C03639=1038.080,62.788,410.793,169.407,39.489,157.422
C03640=1038.074,62.538,410.811,169.405,39.489,157.422
C03641=1038.068,62.289,410.828,169.403,39.488,157.421
C03642=1038.061,62.040,410.846,169.401,39.489,157.421
C03643=1038.055,61.791,410.864,169.399,39.488,157.421
C03644=1038.048,61.541,410.881,169.397,39.488,157.421
C03645=1038.042,61.292,410.899,169.394,39.488,157.421
C03646=1038.035,61.005,410.919,169.392,39.488,157.421
C03647=1038.028,60.719,410.939,169.390,39.487,157.421
C03648=1038.019,60.433,410.959,169.387,39.488,157.421
C03649=1038.012,60.147,410.979,169.385,39.487,157.421
C03650=1038.006,59.897,410.997,169.383,39.487,157.421
C03651=1037.999,59.648,411.014,169.381,39.487,157.420
C03652=1037.994,59.399,411.031,169.379,39.487,157.420
C03653=1037.987,59.150,411.049,169.377,39.487,157.420
C03654=1037.980,58.900,411.066,169.375,39.487,157.420
C03655=1037.974,58.650,411.084,169.373,39.486,157.420
C03656=1037.968,58.402,411.101,169.370,39.486,157.420
C03657=1037.961,58.152,411.118,169.368,39.486,157.420
C03658=1037.955,57.902,411.136,169.366,39.486,157.420
C03659=1037.949,57.654,411.153,169.364,39.486,157.420
C03660=1037.942,57.404,411.171,169.362,39.486,157.419
C03661=1037.936,57.155,411.188,169.360,39.485,157.419
C03662=1037.929,56.906,411.206,169.358,39.485,157.419
C03663=1037.923,56.656,411.223,169.357,39.485,157.419
C03664=1037.917,56.407,411.240,169.355,39.485,157.419
C03665=1037.910,56.158,411.258,169.353,39.485,157.419
C03666=1037.904,55.908,411.276,169.351,39.485,157.419
C03667=1037.898,55.660,411.293,169.349,39.484,157.419
C03668=1037.891,55.410,411.310,169.347,39.484,157.419
C03669=1037.885,55.161,411.328,169.344,39.484,157.419
C03670=1037.878,54.912,411.345,169.342,39.483,157.418
C03671=1037.872,54.662,411.362,169.340,39.484,157.418
C03672=1037.866,54.413,411.380,169.338,39.483,157.418
C03673=1037.860,54.163,411.396,169.336,39.483,157.418
C03674=1037.853,53.914,411.413,169.334,39.483,157.418
C03675=1037.847,53.665,411.431,169.332,39.483,157.418
C03676=1037.840,53.415,411.449,169.330,39.482,157.418
C03677=1037.834,53.166,411.466,169.328,39.483,157.418
C03678=1037.828,52.917,411.484,169.326,39.482,157.418
C03679=1037.822,52.668,411.501,169.324,39.482,157.418
C03680=1037.815,52.418,411.517,169.321,39.482,157.417
C03681=1037.810,52.169,411.535,169.319,39.481,157.417
C03682=1037.803,51.919,411.552,169.317,39.481,157.417
C03683=1037.796,51.671,411.569,169.315,39.481,157.417
C03684=1037.790,51.421,411.587,169.313,39.481,157.417
C03685=1037.784,51.172,411.604,169.311,39.481,157.417
C03686=1037.778,50.922,411.621,169.309,39.481,157.417
C03687=1037.771,50.672,411.639,169.307,39.480,157.417
C03688=1037.765,50.424,411.655,169.305,39.480,157.417
C03689=1037.758,50.174,411.673,169.303,39.480,157.416
C03690=1037.753,49.925,411.690,169.300,39.479,157.416
C03691=1037.746,49.675,411.707,169.298,39.480,157.416
C03692=1037.740,49.427,411.724,169.296,39.479,157.416
C03693=1037.734,49.177,411.742,169.294,39.479,157.416
C03694=1037.728,48.927,411.758,169.293,39.479,157.416
C03695=1037.721,48.678,411.776,169.291,39.478,157.416
C03696=1037.716,48.429,411.793,169.289,39.478,157.416
C03697=1037.709,48.180,411.810,169.287,39.478,157.415
C03698=1037.703,47.930,411.827,169.285,39.478,157.415
C03699=1037.697,47.681,411.844,169.283,39.478,157.415
C03700=1037.690,47.432,411.862,169.280,39.477,157.415
C03701=1037.684,47.182,411.878,169.278,39.477,157.415
C03702=1037.678,46.933,411.896,169.276,39.477,157.415
C03703=1037.672,46.684,411.913,169.274,39.477,157.415
C03704=1037.665,46.434,411.929,169.272,39.476,157.415
C03705=1037.659,46.185,411.946,169.270,39.476,157.415
C03706=1037.653,45.935,411.964,169.268,39.476,157.415
C03707=1037.647,45.686,411.981,169.266,39.476,157.414
C03708=1037.641,45.437,411.998,169.264,39.476,157.414
C03709=1037.635,45.188,412.015,169.262,39.475,157.414
C03710=1037.627,44.901,412.034,169.260,39.475,157.414
C03711=1037.620,44.614,412.054,169.258,39.475,157.414
C03712=1037.613,44.328,412.074,169.254,39.474,157.414
C03713=1037.606,44.042,412.093,169.252,39.474,157.414
C03714=1037.600,43.792,412.110,169.250,39.474,157.414
C03715=1037.594,43.542,412.127,169.248,39.474,157.413
C03716=1037.588,43.293,412.144,169.246,39.473,157.413
C03717=1037.582,43.044,412.161,169.244,39.473,157.413
C03718=1037.575,42.795,412.178,169.242,39.473,157.413
C03719=1037.569,42.545,412.194,169.240,39.473,157.413
C03720=1037.563,42.296,412.211,169.238,39.472,157.413
C03721=1037.556,42.046,412.228,169.236,39.473,157.413
C03722=1037.550,41.797,412.245,169.233,39.472,157.413
C03723=1037.544,41.548,412.261,169.231,39.472,157.413
C03724=1037.537,41.299,412.278,169.229,39.472,157.412
C03725=1037.531,41.049,412.295,169.227,39.472,157.412
C03726=1037.524,40.800,412.312,169.225,39.471,157.412
C03727=1037.518,40.550,412.328,169.223,39.472,157.412
C03728=1037.512,40.302,412.345,169.221,39.471,157.412
C03729=1037.505,40.052,412.362,169.219,39.471,157.412
C03730=1037.499,39.802,412.378,169.217,39.471,157.412
C03731=1037.493,39.553,412.395,169.215,39.471,157.412
C03732=1037.487,39.303,412.412,169.213,39.470,157.412
C03733=1037.481,39.055,412.429,169.211,39.471,157.412
C03734=1037.475,38.804,412.446,169.208,39.470,157.411
C03735=1037.469,38.555,412.462,169.206,39.470,157.411
C03736=1037.462,38.306,412.479,169.204,39.470,157.411
C03737=1037.456,38.056,412.496,169.202,39.470,157.411
C03738=1037.450,37.807,412.512,169.200,39.469,157.411
C03739=1037.444,37.558,412.529,169.198,39.470,157.411
C03740=1037.437,37.308,412.546,169.196,39.469,157.411
C03741=1037.430,37.059,412.561,169.194,39.469,157.411
C03742=1037.424,36.810,412.578,169.192,39.469,157.411
C03743=1037.418,36.560,412.595,169.190,39.469,157.411
C03744=1037.412,36.311,412.611,169.188,39.469,157.411
C03745=1037.405,36.061,412.628,169.186,39.469,157.410
C03746=1037.398,35.813,412.644,169.184,39.469,157.410
C03747=1037.392,35.563,412.660,169.182,39.469,157.410
C03748=1037.386,35.313,412.677,169.179,39.468,157.410
C03749=1037.380,35.064,412.693,169.177,39.469,157.410
C03750=1037.373,34.815,412.710,169.175,39.468,157.410
C03751=1037.366,34.565,412.726,169.173,39.468,157.410
C03752=1037.360,34.316,412.743,169.171,39.468,157.410
C03753=1037.354,34.067,412.759,169.169,39.468,157.410
C03754=1037.348,33.817,412.775,169.167,39.468,157.410
C03755=1037.341,33.568,412.792,169.165,39.468,157.409
C03756=1037.335,33.319,412.808,169.163,39.468,157.409
C03757=1037.329,33.070,412.824,169.161,39.467,157.409
C03758=1037.322,32.819,412.841,169.159,39.467,157.409
C03759=1037.316,32.570,412.857,169.157,39.468,157.409
C03760=1037.309,32.321,412.873,169.155,39.467,157.409
C03761=1037.304,32.072,412.889,169.153,39.467,157.409
C03762=1037.297,31.822,412.906,169.150,39.467,157.409
C03763=1037.291,31.573,412.923,169.147,39.467,157.409
C03764=1037.285,31.324,412.939,169.145,39.466,157.409
C03765=1037.278,31.075,412.955,169.143,39.467,157.409
C03766=1037.272,30.825,412.971,169.141,39.467,157.409
C03767=1037.266,30.575,412.987,169.139,39.466,157.408
C03768=1037.260,30.326,413.004,169.137,39.466,157.408
C03769=1037.253,30.077,413.019,169.135,39.466,157.408
C03770=1037.246,29.827,413.036,169.133,39.466,157.408
C03771=1037.240,29.577,413.052,169.131,39.466,157.408
C03772=1037.234,29.328,413.069,169.129,39.466,157.408
C03773=1037.227,29.080,413.085,169.127,39.466,157.408
C03774=1037.221,28.792,413.104,169.124,39.465,157.408
C03775=1037.213,28.505,413.122,169.121,39.465,157.408
C03776=1037.206,28.219,413.141,169.119,39.465,157.407
C03777=1037.199,27.932,413.159,169.117,39.465,157.407
C03778=1037.193,27.683,413.175,169.115,39.465,157.407
C03779=1037.185,27.433,413.191,169.113,39.465,157.407
C03780=1037.179,27.184,413.208,169.111,39.464,157.407
C03781=1037.174,26.935,413.224,169.109,39.465,157.407
C03782=1037.167,26.686,413.239,169.106,39.465,157.407
C03783=1037.161,26.436,413.256,169.104,39.464,157.407
C03784=1037.154,26.186,413.272,169.102,39.464,157.407
C03785=1037.148,25.937,413.288,169.100,39.465,157.407
C03786=1037.142,25.688,413.304,169.098,39.464,157.407
C03787=1037.135,25.439,413.320,169.096,39.464,157.407
C03788=1037.129,25.189,413.335,169.094,39.464,157.407
C03789=1037.122,24.939,413.351,169.091,39.464,157.406
C03790=1037.116,24.690,413.368,169.089,39.464,157.406
C03791=1037.109,24.441,413.383,169.087,39.464,157.406
C03792=1037.103,24.191,413.400,169.085,39.464,157.406
C03793=1037.097,23.942,413.415,169.083,39.464,157.406
C03794=1037.091,23.693,413.432,169.081,39.464,157.406
C03795=1037.084,23.443,413.447,169.079,39.464,157.406
C03796=1037.078,23.193,413.463,169.076,39.464,157.406
C03797=1037.071,22.944,413.479,169.074,39.464,157.406
C03798=1037.065,22.695,413.495,169.072,39.463,157.406
C03799=1037.059,22.446,413.511,169.070,39.464,157.406
C03800=1037.053,22.196,413.526,169.068,39.463,157.405
C03801=1037.046,21.947,413.542,169.066,39.463,157.405
C03802=1037.040,21.697,413.558,169.064,39.463,157.405
C03803=1037.033,21.448,413.574,169.062,39.463,157.405
C03804=1037.027,21.198,413.590,169.060,39.463,157.405
C03805=1037.021,20.949,413.605,169.057,39.463,157.405
C03806=1037.015,20.699,413.622,169.055,39.463,157.405
C03807=1037.008,20.450,413.637,169.053,39.463,157.405
C03808=1037.002,20.201,413.654,169.051,39.462,157.405
C03809=1036.996,19.951,413.669,169.048,39.463,157.405
C03810=1036.990,19.702,413.685,169.046,39.463,157.405
C03811=1036.983,19.453,413.700,169.044,39.462,157.404
C03812=1036.977,19.202,413.716,169.042,39.462,157.404
C03813=1036.970,18.953,413.732,169.040,39.463,157.404
C03814=1036.963,18.704,413.748,169.038,39.463,157.404
C03815=1036.958,18.454,413.763,169.036,39.462,157.404
C03816=1036.951,18.205,413.779,169.034,39.462,157.404
C03817=1036.945,17.956,413.795,169.032,39.463,157.404
C03818=1036.939,17.706,413.810,169.030,39.462,157.404
C03819=1036.932,17.457,413.826,169.027,39.462,157.404
C03820=1036.926,17.207,413.841,169.025,39.463,157.404
C03821=1036.920,16.958,413.857,169.022,39.462,157.404
C03822=1036.913,16.709,413.873,169.020,39.462,157.404
C03823=1036.907,16.459,413.888,169.018,39.462,157.404
C03824=1036.901,16.210,413.904,169.016,39.462,157.403
C03825=1036.894,15.960,413.919,169.014,39.462,157.403
C03826=1036.888,15.711,413.935,169.012,39.462,157.403
C03827=1036.882,15.462,413.951,169.010,39.462,157.403
C03828=1036.875,15.212,413.966,169.007,39.462,157.403
C03829=1036.869,14.963,413.982,169.005,39.462,157.403
C03830=1036.862,14.713,413.997,169.003,39.462,157.403
C03831=1036.856,14.463,414.013,169.001,39.462,157.403
C03832=1036.850,14.214,414.028,168.999,39.462,157.403
C03833=1036.843,13.965,414.044,168.997,39.462,157.403
C03834=1036.837,13.715,414.059,168.995,39.461,157.403
C03835=1036.830,13.466,414.075,168.993,39.462,157.403
C03836=1036.825,13.216,414.090,168.990,39.462,157.403
C03837=1036.818,12.967,414.106,168.988,39.462,157.403
C03838=1036.811,12.681,414.123,168.986,39.462,157.402
C03839=1036.803,12.396,414.141,168.982,39.462,157.402
C03840=1036.796,12.111,414.158,168.980,39.462,157.402
C03841=1036.789,11.826,414.176,168.977,39.462,157.402
C03842=1036.782,11.576,414.190,168.975,39.462,157.402
C03843=1036.776,11.327,414.205,168.973,39.462,157.402
C03844=1036.769,11.078,414.221,168.971,39.462,157.402
C03845=1036.763,10.828,414.236,168.969,39.462,157.402
C03846=1036.756,10.579,414.252,168.967,39.462,157.402
C03847=1036.750,10.329,414.267,168.964,39.463,157.402
C03848=1036.743,10.080,414.282,168.962,39.463,157.402
C03849=1036.737,9.830,414.298,168.960,39.462,157.402
C03850=1036.731,9.581,414.313,168.958,39.462,157.402
C03851=1036.725,9.331,414.328,168.956,39.462,157.402
C03852=1036.718,9.082,414.343,168.954,39.463,157.402
C03853=1036.712,8.832,414.358,168.952,39.463,157.401
C03854=1036.705,8.583,414.373,168.949,39.462,157.401
C03855=1036.699,8.333,414.388,168.947,39.463,157.401
C03856=1036.692,8.084,414.404,168.945,39.463,157.401
C03857=1036.686,7.834,414.419,168.943,39.463,157.401
C03858=1036.679,7.585,414.434,168.941,39.463,157.401
C03859=1036.673,7.335,414.449,168.938,39.462,157.401
C03860=1036.666,7.086,414.464,168.935,39.463,157.401
C03861=1036.660,6.836,414.479,168.933,39.463,157.401
C03862=1036.655,6.587,414.494,168.931,39.463,157.401
C03863=1036.648,6.337,414.509,168.929,39.463,157.401
C03864=1036.642,6.088,414.525,168.927,39.463,157.401
C03865=1036.635,5.839,414.540,168.925,39.463,157.401
C03866=1036.629,5.589,414.555,168.922,39.463,157.401
C03867=1036.623,5.339,414.570,168.920,39.463,157.400
C03868=1036.616,5.090,414.586,168.918,39.463,157.400
C03869=1036.610,4.841,414.601,168.916,39.463,157.400
C03870=1036.603,4.591,414.615,168.914,39.463,157.400
C03871=1036.597,4.342,414.630,168.912,39.463,157.400
C03872=1036.591,4.092,414.645,168.909,39.463,157.400
C03873=1036.585,3.843,414.660,168.907,39.463,157.400
C03874=1036.578,3.594,414.676,168.905,39.463,157.400
C03875=1036.572,3.344,414.691,168.903,39.463,157.400
C03876=1036.565,3.094,414.706,168.901,39.463,157.400
C03877=1036.559,2.845,414.720,168.898,39.463,157.400
C03878=1036.553,2.596,414.735,168.896,39.463,157.400
C03879=1036.547,2.346,414.750,168.894,39.463,157.400
C03880=1036.540,2.097,414.765,168.892,39.463,157.400
C03881=1036.534,1.847,414.780,168.889,39.463,157.399
C03882=1036.527,1.597,414.795,168.887,39.463,157.399
C03883=1036.521,1.349,414.810,168.884,39.463,157.399
C03884=1036.515,1.099,414.825,168.882,39.463,157.399
C03885=1036.509,0.849,414.841,168.880,39.463,157.399
C03886=1036.503,0.600,414.856,168.878,39.463,157.399
C03887=1036.497,0.350,414.870,168.876,39.463,157.399
C03888=1036.491,0.101,414.885,168.874,39.463,157.399
C03889=1036.484,-0.149,414.900,168.871,39.464,157.399
C03890=1036.478,-0.398,414.915,168.869,39.463,157.399
C03891=1036.472,-0.648,414.930,168.867,39.463,157.399
C03892=1036.466,-0.897,414.944,168.865,39.463,157.399
C03893=1036.460,-1.147,414.959,168.863,39.463,157.399
C03894=1036.453,-1.396,414.974,168.860,39.463,157.398
C03895=1036.447,-1.646,414.989,168.858,39.463,157.398
C03896=1036.441,-1.895,415.004,168.856,39.464,157.398
C03897=1036.435,-2.145,415.019,168.854,39.463,157.398
C03898=1036.428,-2.394,415.034,168.852,39.463,157.398
C03899=1036.422,-2.644,415.049,168.849,39.463,157.398
C03900=1036.416,-2.893,415.063,168.846,39.464,157.398
C03901=1036.410,-3.142,415.078,168.844,39.463,157.398
C03902=1036.399,-3.564,415.103,168.840,39.463,157.398
C03903=1036.388,-3.986,415.128,168.837,39.464,157.398
C03904=1036.380,-4.308,415.147,168.834,39.464,157.398
C03905=1036.372,-4.630,415.165,168.831,39.464,157.398
C03906=1036.364,-4.952,415.184,168.828,39.464,157.398
C03907=1036.355,-5.275,415.203,168.825,39.464,157.397
C03908=1036.349,-5.524,415.217,168.823,39.464,157.397
C03909=1036.342,-5.773,415.232,168.820,39.464,157.397
C03910=1036.336,-6.023,415.246,168.818,39.464,157.397
C03911=1036.330,-6.272,415.261,168.816,39.465,157.397
C03912=1036.323,-6.522,415.275,168.814,39.465,157.397
C03913=1036.317,-6.771,415.290,168.811,39.465,157.397
C03914=1036.311,-7.021,415.304,168.809,39.465,157.397
C03915=1036.304,-7.270,415.318,168.807,39.465,157.397
C03916=1036.298,-7.520,415.333,168.805,39.465,157.397
C03917=1036.291,-7.769,415.348,168.802,39.466,157.397
C03918=1036.285,-8.019,415.361,168.800,39.466,157.397
C03919=1036.279,-8.268,415.376,168.798,39.466,157.397
C03920=1036.272,-8.518,415.391,168.796,39.466,157.397
C03921=1036.266,-8.767,415.404,168.793,39.466,157.397
C03922=1036.260,-9.017,415.419,168.791,39.466,157.397
C03923=1036.253,-9.267,415.434,168.789,39.466,157.397
C03924=1036.247,-9.516,415.448,168.787,39.466,157.397
C03925=1036.241,-9.766,415.463,168.784,39.466,157.397
C03926=1036.234,-10.015,415.478,168.782,39.467,157.396
C03927=1036.228,-10.264,415.491,168.779,39.467,157.396
C03928=1036.222,-10.514,415.506,168.777,39.467,157.396
C03929=1036.215,-10.763,415.520,168.774,39.467,157.396
C03930=1036.209,-11.013,415.534,168.772,39.467,157.396
C03931=1036.203,-11.263,415.549,168.770,39.467,157.396
C03932=1036.196,-11.511,415.563,168.767,39.468,157.396
C03933=1036.190,-11.762,415.577,168.765,39.467,157.396
C03934=1036.185,-12.011,415.592,168.763,39.467,157.396
C03935=1036.178,-12.260,415.605,168.761,39.467,157.396
C03936=1036.171,-12.510,415.620,168.758,39.468,157.396
C03937=1036.166,-12.760,415.634,168.756,39.468,157.396
C03938=1036.159,-13.009,415.648,168.754,39.468,157.396
C03939=1036.153,-13.258,415.663,168.752,39.468,157.396
C03940=1036.146,-13.508,415.677,168.749,39.468,157.396
C03941=1036.140,-13.758,415.692,168.747,39.468,157.396
C03942=1036.134,-14.007,415.706,168.745,39.469,157.396
C03943=1036.127,-14.257,415.720,168.742,39.468,157.395
C03944=1036.122,-14.506,415.734,168.740,39.468,157.395
C03945=1036.115,-14.756,415.749,168.738,39.469,157.395
C03946=1036.109,-15.005,415.762,168.736,39.469,157.395
C03947=1036.103,-15.255,415.777,168.733,39.469,157.395
C03948=1036.096,-15.504,415.790,168.731,39.469,157.395
C03949=1036.090,-15.754,415.805,168.729,39.469,157.395
C03950=1036.084,-16.003,415.818,168.726,39.469,157.395
C03951=1036.078,-16.253,415.833,168.724,39.470,157.395
C03952=1036.071,-16.503,415.847,168.722,39.470,157.395
C03953=1036.064,-16.752,415.860,168.719,39.470,157.395
C03954=1036.058,-17.001,415.875,168.717,39.470,157.395
C03955=1036.052,-17.251,415.888,168.715,39.470,157.395
C03956=1036.045,-17.501,415.902,168.712,39.471,157.395
C03957=1036.039,-17.750,415.917,168.710,39.471,157.395
C03958=1036.032,-18.000,415.930,168.708,39.471,157.395
C03959=1036.027,-18.249,415.944,168.705,39.472,157.395
C03960=1036.020,-18.499,415.959,168.703,39.472,157.395
C03961=1036.014,-18.748,415.972,168.701,39.472,157.395
C03962=1036.008,-18.998,415.986,168.698,39.472,157.395
C03963=1036.001,-19.247,416.000,168.696,39.472,157.395
C03964=1035.994,-19.529,416.015,168.693,39.473,157.395
C03965=1035.986,-19.811,416.031,168.691,39.473,157.395
C03966=1035.980,-20.093,416.047,168.687,39.473,157.394
C03967=1035.972,-20.375,416.063,168.684,39.473,157.394
C03968=1035.966,-20.624,416.076,168.682,39.473,157.394
C03969=1035.960,-20.874,416.090,168.680,39.474,157.394
C03970=1035.953,-21.123,416.104,168.677,39.474,157.394
C03971=1035.947,-21.373,416.118,168.675,39.474,157.394
C03972=1035.941,-21.622,416.132,168.673,39.474,157.394
C03973=1035.934,-21.872,416.145,168.670,39.474,157.394
C03974=1035.928,-22.121,416.160,168.668,39.474,157.394
C03975=1035.922,-22.370,416.173,168.666,39.475,157.394
C03976=1035.915,-22.620,416.187,168.663,39.475,157.394
C03977=1035.910,-22.870,416.201,168.661,39.475,157.394
C03978=1035.903,-23.120,416.214,168.659,39.475,157.394
C03979=1035.897,-23.369,416.228,168.656,39.475,157.394
C03980=1035.891,-23.618,416.242,168.654,39.476,157.394
C03981=1035.884,-23.868,416.256,168.652,39.476,157.394
C03982=1035.878,-24.117,416.269,168.649,39.477,157.394
C03983=1035.872,-24.368,416.283,168.647,39.477,157.394
C03984=1035.866,-24.617,416.296,168.645,39.477,157.394
C03985=1035.860,-24.866,416.310,168.642,39.477,157.394
C03986=1035.853,-25.116,416.325,168.640,39.477,157.394
C03987=1035.847,-25.365,416.338,168.638,39.477,157.394
C03988=1035.841,-25.614,416.351,168.635,39.478,157.394
C03989=1035.834,-25.864,416.365,168.633,39.478,157.394
C03990=1035.829,-26.114,416.379,168.630,39.478,157.393
C03991=1035.822,-26.364,416.392,168.628,39.478,157.393
C03992=1035.815,-26.613,416.406,168.626,39.478,157.393
C03993=1035.810,-26.863,416.419,168.623,39.479,157.393
C03994=1035.803,-27.113,416.433,168.621,39.479,157.393
C03995=1035.797,-27.362,416.446,168.619,39.479,157.393
C03996=1035.791,-27.611,416.460,168.616,39.479,157.393
C03997=1035.784,-27.861,416.473,168.614,39.479,157.393
C03998=1035.778,-28.110,416.487,168.611,39.480,157.393
C03999=1035.772,-28.360,416.500,168.609,39.480,157.393
C04000=1035.765,-28.610,416.514,168.607,39.481,157.393
C04001=1035.759,-28.859,416.527,168.604,39.481,157.393
C04002=1035.752,-29.109,416.541,168.602,39.481,157.393
C04003=1035.746,-29.358,416.554,168.599,39.482,157.393
C04004=1035.740,-29.608,416.568,168.597,39.482,157.393
C04005=1035.733,-29.858,416.581,168.595,39.482,157.393
C04006=1035.727,-30.107,416.594,168.592,39.482,157.393
C04007=1035.721,-30.356,416.608,168.590,39.482,157.393
C04008=1035.715,-30.606,416.620,168.587,39.483,157.393
C04009=1035.708,-30.856,416.634,168.585,39.484,157.393
C04010=1035.702,-31.105,416.647,168.582,39.484,157.393
C04011=1035.696,-31.355,416.660,168.580,39.484,157.393
C04012=1035.689,-31.605,416.674,168.578,39.484,157.393
C04013=1035.683,-31.854,416.687,168.575,39.484,157.393
C04014=1035.676,-32.103,416.701,168.573,39.485,157.393
C04015=1035.670,-32.353,416.713,168.570,39.485,157.393
C04016=1035.664,-32.603,416.727,168.568,39.485,157.393
C04017=1035.658,-32.853,416.741,168.565,39.486,157.393
C04018=1035.652,-33.102,416.754,168.563,39.486,157.393
C04019=1035.646,-33.351,416.767,168.561,39.486,157.393
C04020=1035.639,-33.601,416.781,168.558,39.487,157.393
C04021=1035.633,-33.851,416.793,168.556,39.487,157.393
C04022=1035.627,-34.100,416.807,168.553,39.487,157.393
C04023=1035.621,-34.349,416.820,168.551,39.487,157.392
C04024=1035.614,-34.599,416.834,168.548,39.488,157.392
C04025=1035.608,-34.849,416.846,168.546,39.489,157.393
C04026=1035.602,-35.099,416.859,168.544,39.489,157.392
C04027=1035.595,-35.348,416.873,168.541,39.489,157.392
C04028=1035.588,-35.629,416.887,168.538,39.489,157.392
C04029=1035.581,-35.910,416.903,168.536,39.489,157.392
C04030=1035.574,-36.191,416.917,168.533,39.490,157.392
C04031=1035.567,-36.472,416.931,168.530,39.490,157.392
C04032=1035.561,-36.722,416.945,168.528,39.491,157.392
C04033=1035.555,-36.971,416.958,168.525,39.491,157.392
C04034=1035.549,-37.221,416.970,168.523,39.491,157.392
C04035=1035.542,-37.471,416.984,168.520,39.491,157.392
C04036=1035.536,-37.720,416.997,168.518,39.492,157.392
C04037=1035.530,-37.970,417.010,168.516,39.492,157.392
C04038=1035.524,-38.219,417.023,168.513,39.492,157.392
C04039=1035.517,-38.469,417.036,168.511,39.493,157.392
C04040=1035.511,-38.718,417.049,168.508,39.493,157.392
C04041=1035.505,-38.968,417.063,168.506,39.494,157.392
C04042=1035.499,-39.218,417.075,168.503,39.494,157.392
C04043=1035.492,-39.468,417.088,168.501,39.494,157.392
C04044=1035.486,-39.717,417.102,168.498,39.495,157.392
C04045=1035.480,-39.966,417.114,168.496,39.495,157.392
C04046=1035.473,-40.216,417.127,168.493,39.495,157.392
C04047=1035.467,-40.465,417.139,168.491,39.496,157.392
C04048=1035.461,-40.715,417.153,168.488,39.496,157.392
C04049=1035.454,-40.965,417.165,168.486,39.496,157.392
C04050=1035.448,-41.214,417.178,168.483,39.497,157.392
C04051=1035.442,-41.464,417.191,168.481,39.497,157.392
C04052=1035.436,-41.713,417.204,168.478,39.498,157.392
C04053=1035.429,-41.963,417.216,168.476,39.499,157.392
C04054=1035.423,-42.212,417.229,168.473,39.499,157.392
C04055=1035.417,-42.462,417.242,168.471,39.499,157.392
C04056=1035.411,-42.712,417.254,168.468,39.500,157.392
C04057=1035.403,-42.962,417.268,168.466,39.500,157.392
C04058=1035.398,-43.212,417.280,168.463,39.500,157.392
C04059=1035.391,-43.461,417.293,168.461,39.501,157.392
C04060=1035.385,-43.711,417.306,168.458,39.501,157.392
C04061=1035.378,-43.960,417.319,168.456,39.501,157.392
C04062=1035.373,-44.210,417.331,168.453,39.502,157.392
C04063=1035.367,-44.459,417.344,168.451,39.502,157.392
C04064=1035.360,-44.709,417.357,168.448,39.503,157.392
C04065=1035.354,-44.958,417.369,168.446,39.503,157.392
C04066=1035.348,-45.208,417.381,168.443,39.504,157.392
C04067=1035.342,-45.457,417.395,168.441,39.504,157.392
C04068=1035.336,-45.707,417.407,168.438,39.505,157.392
C04069=1035.329,-45.957,417.419,168.436,39.505,157.392
C04070=1035.323,-46.206,417.433,168.433,39.505,157.392
C04071=1035.317,-46.456,417.445,168.432,39.506,157.392
C04072=1035.310,-46.706,417.457,168.429,39.506,157.392
C04073=1035.304,-46.955,417.470,168.426,39.506,157.392
C04074=1035.298,-47.205,417.483,168.424,39.507,157.392
C04075=1035.292,-47.455,417.495,168.422,39.507,157.392
C04076=1035.285,-47.704,417.508,168.419,39.508,157.392
C04077=1035.279,-47.953,417.521,168.417,39.508,157.392
C04078=1035.274,-48.203,417.533,168.414,39.509,157.392
C04079=1035.267,-48.453,417.545,168.412,39.509,157.392
C04080=1035.261,-48.702,417.558,168.409,39.510,157.392
C04081=1035.255,-48.952,417.571,168.406,39.510,157.392
C04082=1035.248,-49.202,417.583,168.404,39.510,157.392
C04083=1035.242,-49.452,417.595,168.401,39.511,157.392
C04084=1035.236,-49.701,417.609,168.399,39.511,157.392
C04085=1035.230,-49.951,417.621,168.396,39.511,157.391
C04086=1035.223,-50.200,417.633,168.394,39.512,157.392
C04087=1035.218,-50.450,417.646,168.391,39.512,157.392
C04088=1035.211,-50.700,417.658,168.389,39.513,157.391
C04089=1035.206,-50.949,417.670,168.386,39.513,157.392
C04090=1035.199,-51.198,417.682,168.384,39.514,157.392
C04091=1035.193,-51.448,417.695,168.381,39.515,157.392
C04092=1035.185,-51.729,417.708,168.378,39.515,157.392
C04093=1035.178,-52.011,417.722,168.375,39.516,157.392
C04094=1035.171,-52.293,417.736,168.372,39.517,157.392
C04095=1035.163,-52.574,417.749,168.369,39.517,157.392
C04096=1035.157,-52.824,417.762,168.367,39.518,157.392
C04097=1035.151,-53.073,417.774,168.364,39.519,157.392
C04098=1035.144,-53.323,417.786,168.361,39.519,157.392
C04099=1035.138,-53.573,417.798,168.359,39.520,157.392
C04100=1035.132,-53.822,417.810,168.356,39.520,157.392
C04101=1035.125,-54.072,417.822,168.354,39.521,157.392
C04102=1035.119,-54.322,417.835,168.352,39.522,157.392
C04103=1035.112,-54.571,417.847,168.349,39.522,157.392
C04104=1035.106,-54.820,417.858,168.347,39.523,157.392
C04105=1035.100,-55.070,417.871,168.344,39.523,157.392
C04106=1035.094,-55.320,417.883,168.342,39.524,157.392
C04107=1035.087,-55.569,417.895,168.339,39.525,157.392
C04108=1035.081,-55.819,417.907,168.336,39.525,157.392
C04109=1035.075,-56.069,417.919,168.334,39.526,157.392
C04110=1035.068,-56.318,417.931,168.331,39.526,157.392
C04111=1035.062,-56.568,417.944,168.328,39.527,157.392
C04112=1035.056,-56.817,417.955,168.326,39.528,157.392
C04113=1035.050,-57.067,417.967,168.323,39.528,157.392
C04114=1035.044,-57.317,417.979,168.321,39.529,157.392
C04115=1035.037,-57.567,417.991,168.318,39.529,157.392
C04116=1035.030,-57.816,418.003,168.315,39.530,157.392
C04117=1035.025,-58.066,418.016,168.313,39.531,157.392
C04118=1035.018,-58.315,418.027,168.310,39.531,157.392
C04119=1035.012,-58.565,418.039,168.308,39.532,157.392
C04120=1035.006,-58.815,418.050,168.305,39.532,157.392
C04121=1035.000,-59.065,418.063,168.302,39.533,157.392
C04122=1034.993,-59.314,418.075,168.301,39.534,157.392
C04123=1034.987,-59.563,418.087,168.298,39.534,157.392
C04124=1034.981,-59.813,418.099,168.295,39.535,157.392
C04125=1034.975,-60.063,418.110,168.293,39.535,157.392
C04126=1034.968,-60.313,418.122,168.290,39.536,157.392
C04127=1034.961,-60.562,418.134,168.288,39.537,157.392
C04128=1034.956,-60.812,418.146,168.285,39.537,157.392
C04129=1034.949,-61.061,418.158,168.282,39.538,157.392
C04130=1034.943,-61.311,418.170,168.280,39.538,157.392
C04131=1034.937,-61.561,418.182,168.277,39.539,157.392
C04132=1034.931,-61.810,418.194,168.274,39.540,157.392
C04133=1034.925,-62.060,418.205,168.272,39.540,157.392
C04134=1034.918,-62.310,418.217,168.269,39.541,157.392
C04135=1034.913,-62.559,418.229,168.266,39.542,157.392
C04136=1034.906,-62.809,418.241,168.264,39.542,157.392
C04137=1034.900,-63.059,418.252,168.261,39.543,157.392
C04138=1034.893,-63.308,418.264,168.259,39.543,157.392
C04139=1034.888,-63.558,418.277,168.256,39.544,157.392
C04140=1034.882,-63.808,418.288,168.253,39.545,157.392
C04141=1034.875,-64.057,418.300,168.251,39.545,157.392
C04142=1034.869,-64.306,418.311,168.248,39.546,157.392
C04143=1034.863,-64.557,418.323,168.246,39.546,157.393
C04144=1034.857,-64.806,418.335,168.244,39.547,157.393
C04145=1034.851,-65.056,418.346,168.241,39.548,157.393
C04146=1034.844,-65.305,418.358,168.238,39.548,157.393
C04147=1034.838,-65.555,418.371,168.236,39.549,157.393
C04148=1034.833,-65.805,418.381,168.233,39.550,157.393
C04149=1034.826,-66.054,418.393,168.231,39.550,157.393
C04150=1034.820,-66.304,418.405,168.228,39.551,157.393
C04151=1034.814,-66.554,418.417,168.225,39.551,157.393
C04152=1034.808,-66.803,418.429,168.223,39.552,157.393
C04153=1034.802,-67.053,418.440,168.220,39.553,157.393
C04154=1034.795,-67.302,418.452,168.217,39.553,157.393
C04155=1034.790,-67.553,418.463,168.215,39.554,157.393
C04156=1034.783,-67.835,418.476,168.212,39.554,157.393
C04157=1034.776,-68.118,418.489,168.209,39.555,157.393
C04158=1034.769,-68.400,418.503,168.206,39.556,157.393
C04159=1034.762,-68.683,418.516,168.203,39.556,157.393
C04160=1034.756,-68.933,418.527,168.201,39.557,157.393
C04161=1034.749,-69.183,418.539,168.197,39.558,157.393
C04162=1034.744,-69.432,418.550,168.196,39.558,157.393
C04163=1034.737,-69.682,418.562,168.193,39.559,157.393
C04164=1034.732,-69.932,418.574,168.190,39.560,157.393
C04165=1034.726,-70.182,418.585,168.188,39.560,157.393
C04166=1034.720,-70.431,418.596,168.185,39.561,157.393
C04167=1034.713,-70.681,418.608,168.182,39.562,157.393
C04168=1034.707,-70.930,418.619,168.180,39.562,157.393
C04169=1034.702,-71.180,418.631,168.177,39.563,157.393
C04170=1034.696,-71.429,418.643,168.174,39.564,157.393
C04171=1034.689,-71.679,418.654,168.172,39.564,157.393
C04172=1034.683,-71.929,418.665,168.169,39.565,157.393
C04173=1034.677,-72.178,418.677,168.166,39.565,157.393
C04174=1034.672,-72.428,418.688,168.164,39.566,157.393
C04175=1034.666,-72.678,418.700,168.161,39.567,157.393
C04176=1034.659,-72.927,418.711,168.158,39.567,157.393
C04177=1034.653,-73.177,418.722,168.156,39.568,157.393
C04178=1034.647,-73.426,418.734,168.153,39.568,157.393
C04179=1034.641,-73.677,418.746,168.151,39.569,157.393
C04180=1034.636,-73.926,418.757,168.149,39.570,157.393
C04181=1034.629,-74.176,418.768,168.146,39.570,157.393
C04182=1034.623,-74.425,418.780,168.143,39.571,157.393
C04183=1034.617,-74.675,418.791,168.141,39.572,157.393
C04184=1034.611,-74.925,418.802,168.138,39.572,157.393
C04185=1034.605,-75.175,418.813,168.135,39.573,157.393
C04186=1034.598,-75.424,418.824,168.132,39.574,157.393
C04187=1034.592,-75.674,418.835,168.130,39.575,157.394
C04188=1034.586,-75.923,418.846,168.127,39.576,157.394
C04189=1034.580,-76.174,418.857,168.124,39.577,157.394
C04190=1034.574,-76.423,418.868,168.122,39.577,157.394
C04191=1034.568,-76.673,418.879,168.119,39.578,157.394
C04192=1034.562,-76.922,418.891,168.116,39.579,157.394
C04193=1034.556,-77.172,418.902,168.114,39.580,157.394
C04194=1034.550,-77.422,418.913,168.112,39.581,157.394
C04195=1034.544,-77.671,418.924,168.109,39.581,157.394
C04196=1034.537,-77.921,418.935,168.106,39.582,157.394
C04197=1034.531,-78.171,418.945,168.103,39.583,157.394
C04198=1034.525,-78.420,418.956,168.101,39.583,157.394
C04199=1034.519,-78.670,418.968,168.098,39.584,157.394
C04200=1034.513,-78.919,418.979,168.095,39.585,157.394
C04201=1034.506,-79.169,418.990,168.093,39.586,157.394
C04202=1034.501,-79.419,419.001,168.090,39.587,157.394
C04203=1034.495,-79.668,419.012,168.087,39.588,157.394
C04204=1034.489,-79.919,419.023,168.084,39.588,157.394
C04205=1034.482,-80.168,419.034,168.082,39.589,157.394
C04206=1034.476,-80.418,419.045,168.080,39.590,157.394
C04207=1034.470,-80.667,419.056,168.077,39.591,157.394
C04208=1034.464,-80.917,419.066,168.074,39.592,157.394
C04209=1034.457,-81.167,419.077,168.071,39.593,157.395
C04210=1034.452,-81.416,419.088,168.069,39.594,157.395
C04211=1034.444,-81.666,419.099,168.066,39.595,157.395
C04212=1034.439,-81.916,419.110,168.063,39.596,157.395
C04213=1034.433,-82.165,419.121,168.060,39.597,157.395
C04214=1034.426,-82.416,419.131,168.057,39.598,157.395
C04215=1034.420,-82.665,419.141,168.056,39.598,157.395
C04216=1034.414,-82.914,419.152,168.053,39.599,157.395
C04217=1034.408,-83.164,419.163,168.050,39.600,157.395
C04218=1034.402,-83.414,419.174,168.047,39.601,157.395
C04219=1034.395,-83.663,419.184,168.045,39.602,157.395
C04220=1034.388,-83.948,419.196,168.041,39.603,157.395
C04221=1034.381,-84.233,419.208,168.038,39.604,157.395
C04222=1034.374,-84.518,419.221,168.035,39.605,157.395
C04223=1034.367,-84.803,419.233,168.032,39.606,157.396
C04224=1034.361,-85.053,419.244,168.030,39.607,157.396
C04225=1034.355,-85.303,419.255,168.027,39.608,157.396
C04226=1034.349,-85.552,419.265,168.024,39.609,157.396
C04227=1034.343,-85.801,419.276,168.022,39.610,157.396
C04228=1034.336,-86.052,419.286,168.019,39.611,157.396
C04229=1034.331,-86.301,419.297,168.016,39.612,157.396
C04230=1034.325,-86.551,419.308,168.013,39.613,157.396
C04231=1034.318,-86.801,419.318,168.010,39.613,157.396
C04232=1034.312,-87.051,419.328,168.008,39.614,157.396
C04233=1034.306,-87.300,419.339,168.005,39.615,157.396
C04234=1034.300,-87.550,419.350,168.003,39.616,157.396
C04235=1034.294,-87.800,419.361,168.000,39.617,157.396
C04236=1034.288,-88.050,419.370,167.997,39.618,157.396
C04237=1034.282,-88.299,419.381,167.995,39.619,157.397
C04238=1034.275,-88.548,419.392,167.992,39.620,157.397
C04239=1034.270,-88.798,419.402,167.989,39.621,157.397
C04240=1034.264,-89.049,419.413,167.986,39.622,157.397
C04241=1034.257,-89.298,419.423,167.983,39.623,157.397
C04242=1034.251,-89.547,419.434,167.981,39.624,157.397
C04243=1034.245,-89.797,419.444,167.979,39.625,157.397
C04244=1034.239,-90.047,419.455,167.976,39.626,157.397
C04245=1034.232,-90.296,419.465,167.973,39.627,157.397
C04246=1034.227,-90.547,419.475,167.970,39.628,157.397
C04247=1034.221,-90.796,419.486,167.968,39.628,157.397
C04248=1034.215,-91.046,419.496,167.965,39.629,157.397
C04249=1034.209,-91.295,419.507,167.962,39.630,157.397
C04250=1034.203,-91.544,419.517,167.959,39.632,157.397
C04251=1034.197,-91.795,419.527,167.956,39.633,157.397
C04252=1034.190,-92.044,419.538,167.955,39.633,157.398
C04253=1034.185,-92.295,419.548,167.952,39.634,157.398
C04254=1034.179,-92.544,419.559,167.949,39.635,157.398
C04255=1034.173,-92.793,419.569,167.946,39.636,157.398
C04256=1034.167,-93.043,419.579,167.943,39.637,157.398
C04257=1034.161,-93.293,419.590,167.940,39.638,157.398
C04258=1034.155,-93.543,419.600,167.938,39.639,157.398
C04259=1034.149,-93.792,419.610,167.935,39.640,157.398
C04260=1034.143,-94.043,419.620,167.932,39.641,157.398
C04261=1034.136,-94.292,419.631,167.930,39.642,157.398
C04262=1034.131,-94.542,419.641,167.927,39.643,157.398
C04263=1034.125,-94.791,419.652,167.925,39.644,157.398
C04264=1034.119,-95.041,419.661,167.922,39.645,157.398
C04265=1034.113,-95.291,419.672,167.919,39.646,157.398
C04266=1034.107,-95.540,419.682,167.916,39.647,157.398
C04267=1034.101,-95.790,419.693,167.913,39.648,157.398
C04268=1034.095,-96.040,419.702,167.911,39.648,157.399
C04269=1034.089,-96.289,419.713,167.908,39.650,157.399
C04270=1034.083,-96.539,419.723,167.906,39.651,157.399
C04271=1034.078,-96.789,419.733,167.903,39.652,157.399
C04272=1034.071,-97.038,419.743,167.900,39.653,157.399
C04273=1034.066,-97.288,419.753,167.897,39.654,157.399
C04274=1034.059,-97.538,419.764,167.895,39.655,157.399
C04275=1034.054,-97.788,419.774,167.892,39.655,157.399
C04276=1034.048,-98.038,419.783,167.889,39.657,157.399
C04277=1034.041,-98.287,419.794,167.886,39.658,157.399
C04278=1034.035,-98.538,419.804,167.883,39.659,157.399
C04279=1034.029,-98.787,419.814,167.881,39.660,157.400
C04280=1034.023,-99.037,419.824,167.878,39.661,157.400
C04281=1034.016,-99.286,419.834,167.876,39.662,157.400
C04282=1034.011,-99.536,419.844,167.873,39.664,157.400
C04283=1034.005,-99.786,419.853,167.870,39.665,157.400
C04284=1033.998,-100.073,419.864,167.866,39.666,157.400
C04285=1033.991,-100.360,419.877,167.864,39.667,157.400
C04286=1033.984,-100.647,419.888,167.861,39.668,157.400
C04287=1033.977,-100.934,419.899,167.858,39.670,157.400
C04288=1033.971,-101.184,419.908,167.855,39.671,157.400
C04289=1033.966,-101.434,419.919,167.852,39.672,157.401
C04290=1033.959,-101.683,419.928,167.849,39.673,157.401
C04291=1033.953,-101.933,419.938,167.846,39.674,157.401
C04292=1033.947,-102.182,419.948,167.844,39.676,157.401
C04293=1033.941,-102.433,419.958,167.841,39.677,157.401
C04294=1033.935,-102.682,419.968,167.838,39.677,157.401
C04295=1033.929,-102.932,419.977,167.836,39.679,157.401
C04296=1033.923,-103.181,419.988,167.833,39.680,157.401
C04297=1033.917,-103.431,419.998,167.830,39.681,157.401
C04298=1033.911,-103.681,420.007,167.827,39.682,157.401
C04299=1033.905,-103.931,420.017,167.825,39.683,157.401
C04300=1033.899,-104.181,420.026,167.822,39.684,157.401
C04301=1033.893,-104.431,420.037,167.819,39.686,157.402
C04302=1033.888,-104.680,420.046,167.816,39.687,157.402
C04303=1033.881,-104.930,420.055,167.813,39.688,157.402
C04304=1033.875,-105.180,420.065,167.811,39.689,157.402
C04305=1033.869,-105.429,420.074,167.808,39.690,157.402
C04306=1033.863,-105.679,420.085,167.806,39.692,157.402
C04307=1033.857,-105.929,420.095,167.803,39.693,157.402
C04308=1033.851,-106.179,420.104,167.800,39.693,157.402
C04309=1033.845,-106.428,420.114,167.797,39.695,157.402
C04310=1033.839,-106.677,420.123,167.794,39.696,157.402
C04311=1033.833,-106.927,420.133,167.791,39.698,157.403
C04312=1033.828,-107.177,420.143,167.788,39.698,157.403
C04313=1033.822,-107.427,420.153,167.787,39.699,157.403
C04314=1033.815,-107.677,420.162,167.784,39.701,157.403
C04315=1033.809,-107.927,420.172,167.781,39.702,157.403
C04316=1033.803,-108.177,420.181,167.778,39.703,157.403
C04317=1033.798,-108.426,420.190,167.775,39.704,157.403
C04318=1033.792,-108.676,420.199,167.772,39.706,157.403
C04319=1033.785,-108.926,420.209,167.770,39.707,157.403
C04320=1033.779,-109.176,420.218,167.767,39.708,157.404
C04321=1033.773,-109.425,420.228,167.764,39.709,157.404
C04322=1033.767,-109.675,420.238,167.761,39.711,157.404
C04323=1033.761,-109.924,420.247,167.758,39.712,157.404
C04324=1033.755,-110.174,420.256,167.755,39.713,157.404
C04325=1033.749,-110.424,420.266,167.753,39.714,157.404
C04326=1033.743,-110.674,420.275,167.751,39.716,157.404
C04327=1033.737,-110.924,420.284,167.748,39.717,157.404
C04328=1033.731,-111.173,420.294,167.745,39.718,157.404
C04329=1033.725,-111.423,420.303,167.742,39.719,157.405
C04330=1033.719,-111.673,420.313,167.739,39.721,157.405
C04331=1033.713,-111.923,420.322,167.736,39.722,157.405
C04332=1033.708,-112.172,420.331,167.734,39.723,157.405
C04333=1033.701,-112.422,420.340,167.731,39.725,157.405
C04334=1033.695,-112.672,420.350,167.728,39.726,157.405
C04335=1033.689,-112.922,420.359,167.725,39.727,157.405
C04336=1033.683,-113.171,420.369,167.722,39.728,157.405
C04337=1033.678,-113.421,420.377,167.720,39.730,157.406
C04338=1033.671,-113.671,420.387,167.718,39.731,157.406
C04339=1033.666,-113.920,420.396,167.715,39.732,157.406
C04340=1033.660,-114.171,420.405,167.712,39.733,157.406
C04341=1033.654,-114.420,420.415,167.709,39.735,157.406
C04342=1033.648,-114.670,420.424,167.706,39.736,157.406
C04343=1033.642,-114.919,420.433,167.704,39.737,157.406
C04344=1033.636,-115.170,420.442,167.701,39.739,157.406
C04345=1033.630,-115.419,420.452,167.698,39.740,157.406
C04346=1033.624,-115.669,420.461,167.695,39.741,157.407
C04347=1033.619,-115.919,420.470,167.692,39.743,157.407
C04348=1033.611,-116.205,420.480,167.689,39.744,157.407
C04349=1033.604,-116.492,420.491,167.686,39.746,157.407
C04350=1033.598,-116.778,420.502,167.683,39.747,157.407
C04351=1033.591,-117.065,420.511,167.680,39.749,157.407
C04352=1033.585,-117.315,420.521,167.677,39.750,157.407
C04353=1033.579,-117.564,420.530,167.674,39.751,157.408
C04354=1033.574,-117.814,420.539,167.672,39.753,157.408
C04355=1033.567,-118.064,420.548,167.669,39.755,157.408
C04356=1033.562,-118.314,420.557,167.666,39.755,157.408
C04357=1033.555,-118.563,420.566,167.663,39.757,157.408
C04358=1033.549,-118.813,420.575,167.660,39.759,157.408
C04359=1033.543,-119.063,420.584,167.657,39.760,157.408
C04360=1033.538,-119.312,420.593,167.655,39.761,157.408
C04361=1033.532,-119.563,420.602,167.652,39.763,157.409
C04362=1033.525,-119.812,420.611,167.649,39.764,157.409
C04363=1033.520,-120.062,420.620,167.646,39.765,157.409
C04364=1033.513,-120.312,420.629,167.643,39.767,157.409
C04365=1033.508,-120.561,420.638,167.641,39.768,157.409
C04366=1033.502,-120.812,420.647,167.638,39.769,157.409
C04367=1033.497,-121.061,420.656,167.635,39.771,157.409
C04368=1033.490,-121.311,420.664,167.632,39.773,157.410
C04369=1033.484,-121.561,420.674,167.629,39.774,157.410
C04370=1033.479,-121.811,420.682,167.627,39.775,157.410
C04371=1033.473,-122.060,420.692,167.624,39.777,157.410
C04372=1033.467,-122.310,420.700,167.621,39.778,157.410
C04373=1033.460,-122.560,420.709,167.618,39.779,157.410
C04374=1033.455,-122.809,420.718,167.615,39.781,157.410
C04375=1033.449,-123.060,420.726,167.613,39.782,157.410
C04376=1033.443,-123.309,420.735,167.610,39.784,157.411
C04377=1033.437,-123.559,420.744,167.608,39.785,157.411
C04378=1033.432,-123.809,420.752,167.605,39.786,157.411
C04379=1033.426,-124.058,420.762,167.602,39.788,157.411
C04380=1033.420,-124.308,420.770,167.600,39.790,157.411
C04381=1033.414,-124.558,420.779,167.597,39.791,157.411
C04382=1033.408,-124.807,420.788,167.594,39.792,157.411
C04383=1033.402,-125.057,420.796,167.591,39.794,157.412
C04384=1033.396,-125.307,420.805,167.588,39.795,157.412
C04385=1033.390,-125.557,420.814,167.586,39.797,157.412
C04386=1033.384,-125.806,420.822,167.583,39.799,157.412
C04387=1033.378,-126.057,420.831,167.580,39.800,157.412
C04388=1033.372,-126.306,420.839,167.577,39.801,157.412
C04389=1033.366,-126.556,420.848,167.574,39.803,157.412
C04390=1033.361,-126.806,420.857,167.572,39.804,157.413
C04391=1033.354,-127.056,420.865,167.569,39.806,157.413
C04392=1033.349,-127.306,420.874,167.566,39.808,157.413
C04393=1033.342,-127.555,420.883,167.563,39.809,157.413
C04394=1033.337,-127.805,420.891,167.560,39.811,157.413
C04395=1033.332,-128.054,420.900,167.558,39.812,157.413
C04396=1033.327,-128.304,420.909,167.555,39.813,157.413
C04397=1033.323,-128.554,420.920,167.553,39.813,157.413
C04398=1033.319,-128.804,420.931,167.549,39.812,157.413
C04399=1033.316,-129.053,420.941,167.547,39.812,157.413
C04400=1033.315,-129.304,420.954,167.545,39.811,157.413
C04401=1033.313,-129.553,420.966,167.543,39.809,157.412
C04402=1033.312,-129.803,420.979,167.541,39.807,157.412
C04403=1033.312,-130.053,420.993,167.539,39.805,157.412
C04404=1033.313,-130.303,421.007,167.537,39.802,157.411
C04405=1033.315,-130.553,421.022,167.535,39.798,157.410
C04406=1033.316,-130.802,421.037,167.534,39.794,157.410
C04407=1033.320,-131.052,421.053,167.533,39.790,157.409
C04408=1033.322,-131.303,421.070,167.531,39.786,157.408
C04409=1033.327,-131.553,421.086,167.530,39.780,157.407
C04410=1033.331,-131.802,421.105,167.529,39.775,157.406
C04411=1033.337,-132.053,421.122,167.528,39.768,157.405
C04412=1033.008,-132.077,420.834,167.479,39.995,157.441
C04413=1033.002,-131.827,420.816,167.480,40.001,157.442
C04414=1032.998,-131.578,420.797,167.481,40.006,157.443
C04415=1032.994,-131.327,420.780,167.482,40.011,157.444
C04416=1032.991,-131.077,420.764,167.483,40.016,157.445
C04417=1032.988,-130.828,420.748,167.485,40.021,157.446
C04418=1032.986,-130.578,420.733,167.487,40.025,157.446
C04419=1032.984,-130.327,420.718,167.489,40.028,157.447
C04420=1032.984,-130.077,420.704,167.490,40.031,157.447
C04421=1032.984,-129.827,420.690,167.493,40.033,157.448
C04422=1032.985,-129.577,420.677,167.494,40.035,157.448
C04423=1032.986,-129.328,420.664,167.497,40.037,157.449
C04424=1032.988,-129.078,420.653,167.499,40.038,157.449
C04425=1032.991,-128.828,420.642,167.501,40.039,157.449
C04426=1032.994,-128.579,420.631,167.503,40.039,157.449
C04427=1032.998,-128.329,420.621,167.506,40.038,157.449
C04428=1033.003,-128.079,420.611,167.508,40.038,157.449
C04429=1033.008,-127.830,420.602,167.511,40.037,157.449
C04430=1033.014,-127.579,420.594,167.514,40.035,157.449
C04431=1033.020,-127.331,420.585,167.517,40.033,157.449
C04432=1033.025,-127.081,420.576,167.519,40.032,157.449
C04433=1033.031,-126.830,420.568,167.522,40.030,157.449
C04434=1033.037,-126.582,420.559,167.525,40.029,157.449
C04435=1033.043,-126.331,420.550,167.528,40.028,157.448
C04436=1033.049,-126.082,420.542,167.531,40.026,157.448
C04437=1033.055,-125.831,420.533,167.533,40.024,157.448
C04438=1033.061,-125.582,420.524,167.537,40.023,157.448
C04439=1033.067,-125.332,420.516,167.540,40.021,157.448
C04440=1033.073,-125.082,420.507,167.543,40.019,157.448
C04441=1033.078,-124.832,420.499,167.545,40.018,157.447
C04442=1033.085,-124.583,420.490,167.548,40.016,157.447
C04443=1033.091,-124.333,420.481,167.551,40.014,157.447
C04444=1033.096,-124.083,420.473,167.554,40.014,157.447
C04445=1033.103,-123.834,420.464,167.557,40.012,157.447
C04446=1033.108,-123.584,420.455,167.559,40.010,157.447
C04447=1033.114,-123.334,420.446,167.562,40.009,157.447
C04448=1033.120,-123.084,420.437,167.565,40.008,157.447
C04449=1033.126,-122.834,420.429,167.568,40.006,157.446
C04450=1033.131,-122.585,420.420,167.571,40.005,157.446
C04451=1033.138,-122.335,420.411,167.573,40.003,157.446
C04452=1033.143,-122.085,420.402,167.576,40.001,157.446
C04453=1033.150,-121.836,420.393,167.578,40.000,157.446
C04454=1033.155,-121.586,420.385,167.581,39.999,157.446
C04455=1033.161,-121.336,420.375,167.584,39.997,157.446
C04456=1033.167,-121.086,420.366,167.586,39.996,157.445
C04457=1033.173,-120.836,420.359,167.589,39.995,157.445
C04458=1033.179,-120.586,420.349,167.592,39.993,157.445
C04459=1033.185,-120.337,420.341,167.595,39.991,157.445
C04460=1033.191,-120.087,420.331,167.598,39.990,157.445
C04461=1033.196,-119.837,420.322,167.600,39.989,157.445
C04462=1033.202,-119.587,420.313,167.603,39.987,157.445
C04463=1033.209,-119.337,420.305,167.606,39.986,157.444
C04464=1033.214,-119.088,420.295,167.609,39.984,157.444
C04465=1033.220,-118.838,420.287,167.612,39.983,157.444
C04466=1033.226,-118.588,420.277,167.614,39.981,157.444
C04467=1033.232,-118.338,420.269,167.617,39.980,157.444
C04468=1033.238,-118.089,420.260,167.620,39.978,157.444
C04469=1033.244,-117.839,420.251,167.623,39.977,157.444
C04470=1033.250,-117.589,420.242,167.626,39.976,157.444
C04471=1033.256,-117.340,420.232,167.628,39.974,157.443
C04472=1033.261,-117.090,420.223,167.631,39.973,157.443
C04473=1033.269,-116.803,420.213,167.635,39.971,157.443
C04474=1033.276,-116.517,420.202,167.638,39.970,157.443
C04475=1033.282,-116.230,420.191,167.641,39.968,157.443
C04476=1033.289,-115.943,420.182,167.644,39.967,157.443
C04477=1033.295,-115.694,420.173,167.647,39.965,157.443
C04478=1033.301,-115.444,420.163,167.650,39.963,157.442
C04479=1033.307,-115.194,420.154,167.653,39.962,157.442
C04480=1033.313,-114.945,420.145,167.656,39.961,157.442
C04481=1033.319,-114.695,420.135,167.658,39.959,157.442
C04482=1033.325,-114.445,420.127,167.661,39.958,157.442
C04483=1033.330,-114.196,420.117,167.664,39.957,157.442
C04484=1033.336,-113.946,420.108,167.667,39.956,157.442
C04485=1033.342,-113.695,420.099,167.669,39.954,157.442
C04486=1033.348,-113.446,420.089,167.671,39.953,157.441
C04487=1033.354,-113.197,420.080,167.674,39.952,157.441
C04488=1033.360,-112.947,420.071,167.677,39.950,157.441
C04489=1033.366,-112.696,420.062,167.680,39.949,157.441
C04490=1033.372,-112.447,420.053,167.683,39.947,157.441
C04491=1033.378,-112.197,420.043,167.686,39.946,157.441
C04492=1033.384,-111.948,420.034,167.688,39.945,157.441
C04493=1033.390,-111.698,420.024,167.691,39.943,157.441
C04494=1033.395,-111.448,420.015,167.694,39.942,157.441
C04495=1033.402,-111.198,420.006,167.697,39.941,157.440
C04496=1033.408,-110.949,419.996,167.700,39.940,157.440
C04497=1033.414,-110.699,419.987,167.703,39.938,157.440
C04498=1033.420,-110.449,419.977,167.705,39.937,157.440
C04499=1033.426,-110.200,419.968,167.708,39.936,157.440
C04500=1033.431,-109.949,419.959,167.711,39.934,157.440
C04501=1033.438,-109.700,419.950,167.714,39.933,157.440
C04502=1033.444,-109.450,419.940,167.717,39.932,157.440
C04503=1033.450,-109.200,419.930,167.720,39.931,157.440
C04504=1033.456,-108.951,419.921,167.721,39.929,157.439
C04505=1033.462,-108.701,419.912,167.724,39.928,157.439
C04506=1033.468,-108.451,419.902,167.727,39.927,157.439
C04507=1033.474,-108.202,419.893,167.730,39.926,157.439
C04508=1033.480,-107.952,419.883,167.733,39.924,157.439
C04509=1033.486,-107.702,419.873,167.735,39.922,157.439
C04510=1033.492,-107.453,419.864,167.738,39.921,157.439
C04511=1033.498,-107.202,419.855,167.741,39.920,157.439
C04512=1033.503,-106.952,419.845,167.744,39.919,157.439
C04513=1033.509,-106.703,419.836,167.747,39.918,157.438
C04514=1033.516,-106.453,419.826,167.750,39.916,157.438
C04515=1033.522,-106.203,419.816,167.753,39.915,157.438
C04516=1033.528,-105.954,419.807,167.755,39.914,157.438
C04517=1033.534,-105.705,419.797,167.758,39.913,157.438
C04518=1033.539,-105.455,419.787,167.760,39.911,157.438
C04519=1033.545,-105.205,419.777,167.763,39.910,157.438
C04520=1033.552,-104.955,419.768,167.766,39.909,157.438
C04521=1033.558,-104.705,419.758,167.769,39.908,157.438
C04522=1033.564,-104.455,419.749,167.772,39.907,157.438
C04523=1033.569,-104.205,419.738,167.774,39.905,157.437
C04524=1033.576,-103.955,419.729,167.777,39.904,157.437
C04525=1033.581,-103.706,419.720,167.780,39.903,157.437
C04526=1033.587,-103.457,419.710,167.783,39.902,157.437
C04527=1033.593,-103.206,419.700,167.786,39.901,157.437
C04528=1033.599,-102.957,419.690,167.788,39.899,157.437
C04529=1033.605,-102.707,419.680,167.790,39.899,157.437
C04530=1033.612,-102.458,419.670,167.793,39.897,157.437
C04531=1033.617,-102.208,419.660,167.796,39.896,157.437
C04532=1033.623,-101.958,419.651,167.799,39.895,157.437
C04533=1033.629,-101.708,419.641,167.802,39.893,157.436
C04534=1033.636,-101.459,419.631,167.805,39.893,157.436
C04535=1033.641,-101.209,419.621,167.808,39.892,157.436
C04536=1033.647,-100.959,419.611,167.810,39.890,157.436
C04537=1033.654,-100.672,419.600,167.813,39.889,157.436
C04538=1033.661,-100.385,419.589,167.816,39.887,157.436
C04539=1033.668,-100.097,419.577,167.820,39.886,157.436
C04540=1033.675,-99.811,419.566,167.823,39.885,157.436
C04541=1033.681,-99.562,419.556,167.825,39.883,157.436
C04542=1033.687,-99.312,419.547,167.828,39.882,157.436
C04543=1033.693,-99.062,419.536,167.831,39.881,157.435
C04544=1033.699,-98.812,419.526,167.834,39.880,157.435
C04545=1033.705,-98.563,419.517,167.836,39.879,157.435
C04546=1033.711,-98.312,419.506,167.839,39.878,157.435
C04547=1033.718,-98.062,419.496,167.842,39.876,157.435
C04548=1033.724,-97.813,419.486,167.844,39.876,157.435
C04549=1033.730,-97.563,419.477,167.847,39.875,157.435
C04550=1033.736,-97.313,419.466,167.850,39.873,157.435
C04551=1033.741,-97.063,419.456,167.853,39.872,157.435
C04552=1033.748,-96.814,419.446,167.856,39.871,157.435
C04553=1033.753,-96.564,419.435,167.858,39.870,157.435
C04554=1033.760,-96.314,419.426,167.861,39.869,157.435
C04555=1033.765,-96.064,419.415,167.864,39.868,157.434
C04556=1033.771,-95.815,419.405,167.866,39.867,157.434
C04557=1033.777,-95.565,419.395,167.869,39.866,157.434
C04558=1033.783,-95.316,419.385,167.872,39.865,157.434
C04559=1033.789,-95.066,419.374,167.874,39.864,157.434
C04560=1033.795,-94.816,419.364,167.877,39.863,157.434
C04561=1033.801,-94.566,419.354,167.880,39.862,157.434
C04562=1033.807,-94.317,419.344,167.883,39.861,157.434
C04563=1033.813,-94.067,419.334,167.886,39.860,157.434
C04564=1033.819,-93.818,419.323,167.888,39.859,157.434
C04565=1033.825,-93.568,419.313,167.890,39.858,157.434
C04566=1033.831,-93.318,419.302,167.893,39.857,157.434
C04567=1033.837,-93.068,419.292,167.896,39.856,157.434
C04568=1033.843,-92.818,419.281,167.899,39.855,157.433
C04569=1033.849,-92.569,419.272,167.902,39.854,157.433
C04570=1033.855,-92.319,419.261,167.905,39.853,157.433
C04571=1033.861,-92.070,419.251,167.907,39.852,157.433
C04572=1033.867,-91.820,419.241,167.910,39.851,157.433
C04573=1033.873,-91.571,419.230,167.912,39.850,157.433
C04574=1033.879,-91.320,419.220,167.915,39.849,157.433
C04575=1033.885,-91.070,419.209,167.918,39.847,157.433
C04576=1033.891,-90.821,419.199,167.921,39.847,157.433
C04577=1033.897,-90.571,419.188,167.923,39.846,157.433
C04578=1033.903,-90.322,419.178,167.926,39.845,157.433
C04579=1033.909,-90.072,419.168,167.929,39.844,157.433
C04580=1033.916,-89.822,419.157,167.932,39.843,157.433
C04581=1033.922,-89.572,419.146,167.935,39.842,157.433
C04582=1033.927,-89.322,419.136,167.937,39.841,157.433
C04583=1033.933,-89.073,419.126,167.939,39.840,157.432
C04584=1033.939,-88.824,419.115,167.942,39.839,157.432
C04585=1033.946,-88.573,419.105,167.945,39.838,157.432
C04586=1033.952,-88.324,419.094,167.948,39.837,157.432
C04587=1033.957,-88.074,419.083,167.951,39.836,157.432
C04588=1033.964,-87.825,419.073,167.954,39.835,157.432
C04589=1033.969,-87.575,419.063,167.956,39.834,157.432
C04590=1033.976,-87.325,419.052,167.958,39.833,157.432
C04591=1033.982,-87.075,419.041,167.961,39.832,157.432
C04592=1033.988,-86.825,419.031,167.964,39.831,157.432
C04593=1033.994,-86.576,419.021,167.967,39.830,157.432
C04594=1034.000,-86.326,419.010,167.970,39.829,157.432
C04595=1034.007,-86.077,419.000,167.972,39.828,157.432
C04596=1034.013,-85.827,418.989,167.975,39.827,157.432
C04597=1034.018,-85.577,418.978,167.978,39.826,157.432
C04598=1034.025,-85.327,418.968,167.981,39.825,157.431
C04599=1034.031,-85.078,418.957,167.983,39.824,157.431
C04600=1034.037,-84.829,418.947,167.985,39.823,157.431
C04601=1034.045,-84.543,418.934,167.989,39.822,157.431
C04602=1034.051,-84.259,418.922,167.992,39.821,157.431
C04603=1034.059,-83.973,418.910,167.995,39.820,157.431
C04604=1034.065,-83.689,418.898,167.998,39.818,157.431
C04605=1034.071,-83.439,418.887,168.001,39.817,157.431
C04606=1034.078,-83.189,418.876,168.003,39.817,157.431
C04607=1034.084,-82.940,418.866,168.006,39.816,157.431
C04608=1034.090,-82.690,418.855,168.009,39.815,157.431
C04609=1034.096,-82.440,418.844,168.011,39.814,157.431
C04610=1034.102,-82.190,418.834,168.014,39.813,157.431
C04611=1034.108,-81.941,418.823,168.017,39.812,157.431
C04612=1034.115,-81.691,418.813,168.020,39.810,157.430
C04613=1034.121,-81.441,418.802,168.023,39.809,157.430
C04614=1034.127,-81.191,418.790,168.025,39.809,157.430
C04615=1034.134,-80.942,418.780,168.027,39.808,157.430
C04616=1034.139,-80.693,418.769,168.030,39.807,157.430
C04617=1034.146,-80.442,418.758,168.033,39.806,157.430
C04618=1034.152,-80.193,418.748,168.036,39.805,157.430
C04619=1034.159,-79.943,418.737,168.038,39.804,157.430
C04620=1034.164,-79.694,418.726,168.041,39.803,157.430
C04621=1034.170,-79.444,418.715,168.044,39.802,157.430
C04622=1034.176,-79.194,418.704,168.047,39.801,157.430
C04623=1034.182,-78.944,418.693,168.049,39.801,157.430
C04624=1034.189,-78.695,418.682,168.052,39.800,157.430
C04625=1034.195,-78.445,418.671,168.054,39.799,157.430
C04626=1034.201,-78.195,418.660,168.057,39.798,157.430
C04627=1034.207,-77.946,418.648,168.059,39.798,157.430
C04628=1034.213,-77.696,418.637,168.062,39.797,157.430
C04629=1034.219,-77.446,418.626,168.065,39.796,157.430
C04630=1034.225,-77.197,418.615,168.068,39.795,157.429
C04631=1034.231,-76.947,418.604,168.070,39.794,157.429
C04632=1034.237,-76.697,418.593,168.073,39.793,157.429
C04633=1034.243,-76.448,418.582,168.076,39.792,157.429
C04634=1034.250,-76.198,418.571,168.079,39.791,157.429
C04635=1034.256,-75.949,418.560,168.081,39.790,157.429
C04636=1034.262,-75.699,418.549,168.083,39.790,157.429
C04637=1034.268,-75.449,418.538,168.086,39.789,157.429
C04638=1034.274,-75.199,418.527,168.089,39.788,157.429
C04639=1034.281,-74.950,418.515,168.091,39.788,157.429
C04640=1034.287,-74.700,418.504,168.094,39.787,157.429
C04641=1034.293,-74.450,418.493,168.097,39.786,157.429
C04642=1034.299,-74.200,418.482,168.100,39.785,157.429
C04643=1034.305,-73.951,418.471,168.102,39.784,157.429
C04644=1034.311,-73.702,418.459,168.105,39.784,157.429
C04645=1034.317,-73.452,418.448,168.108,39.783,157.429
C04646=1034.323,-73.202,418.437,168.110,39.782,157.429
C04647=1034.329,-72.952,418.425,168.113,39.781,157.429
C04648=1034.334,-72.703,418.414,168.116,39.781,157.429
C04649=1034.341,-72.453,418.402,168.119,39.780,157.429
C04650=1034.347,-72.204,418.391,168.120,39.779,157.429
C04651=1034.353,-71.954,418.380,168.123,39.779,157.429
C04652=1034.358,-71.704,418.367,168.126,39.778,157.429
C04653=1034.365,-71.454,418.356,168.128,39.777,157.429
C04654=1034.371,-71.205,418.345,168.131,39.777,157.429
C04655=1034.377,-70.955,418.333,168.134,39.776,157.429
C04656=1034.383,-70.706,418.322,168.136,39.775,157.429
C04657=1034.390,-70.456,418.311,168.139,39.774,157.428
C04658=1034.395,-70.206,418.299,168.142,39.774,157.429
C04659=1034.401,-69.956,418.288,168.144,39.773,157.428
C04660=1034.407,-69.707,418.276,168.147,39.772,157.428
C04661=1034.413,-69.457,418.265,168.150,39.772,157.429
C04662=1034.419,-69.207,418.252,168.152,39.771,157.428
C04663=1034.425,-68.958,418.242,168.155,39.770,157.428
C04664=1034.432,-68.708,418.230,168.158,39.770,157.428
C04665=1034.438,-68.425,418.217,168.161,39.769,157.428
C04666=1034.445,-68.143,418.204,168.163,39.768,157.428
C04667=1034.452,-67.860,418.191,168.166,39.767,157.428
C04668=1034.459,-67.577,418.178,168.169,39.766,157.428
C04669=1034.465,-67.328,418.166,168.172,39.766,157.428
C04670=1034.472,-67.078,418.154,168.174,39.765,157.428
C04671=1034.477,-66.828,418.142,168.177,39.764,157.428
C04672=1034.483,-66.578,418.131,168.180,39.764,157.428
C04673=1034.489,-66.329,418.119,168.182,39.763,157.428
C04674=1034.496,-66.079,418.108,168.185,39.762,157.428
C04675=1034.502,-65.829,418.096,168.188,39.762,157.428
C04676=1034.508,-65.580,418.084,168.190,39.761,157.428
C04677=1034.514,-65.330,418.073,168.193,39.760,157.428
C04678=1034.521,-65.081,418.061,168.196,39.760,157.428
C04679=1034.526,-64.831,418.050,168.198,39.759,157.428
C04680=1034.532,-64.581,418.037,168.201,39.758,157.428
C04681=1034.539,-64.332,418.025,168.204,39.758,157.428
C04682=1034.545,-64.082,418.015,168.205,39.757,157.428
C04683=1034.551,-63.833,418.003,168.208,39.756,157.428
C04684=1034.557,-63.583,417.990,168.211,39.756,157.428
C04685=1034.563,-63.333,417.979,168.213,39.755,157.428
C04686=1034.570,-63.084,417.967,168.216,39.754,157.428
C04687=1034.575,-62.834,417.955,168.219,39.754,157.428
C04688=1034.581,-62.584,417.944,168.221,39.753,157.428
C04689=1034.588,-62.335,417.932,168.224,39.752,157.428
C04690=1034.594,-62.085,417.920,168.226,39.752,157.428
C04691=1034.600,-61.835,417.908,168.229,39.751,157.428
C04692=1034.606,-61.586,417.896,168.232,39.750,157.428
C04693=1034.613,-61.336,417.884,168.234,39.750,157.428
C04694=1034.619,-61.087,417.872,168.237,39.749,157.428
C04695=1034.625,-60.836,417.861,168.240,39.748,157.428
C04696=1034.631,-60.587,417.849,168.242,39.747,157.428
C04697=1034.638,-60.338,417.837,168.245,39.747,157.428
C04698=1034.644,-60.088,417.825,168.248,39.746,157.428
C04699=1034.650,-59.838,417.813,168.249,39.745,157.428
C04700=1034.656,-59.589,417.802,168.252,39.745,157.428
C04701=1034.663,-59.339,417.790,168.255,39.744,157.428
C04702=1034.669,-59.089,417.777,168.257,39.743,157.427
C04703=1034.675,-58.840,417.765,168.260,39.743,157.428
C04704=1034.682,-58.590,417.754,168.263,39.742,157.427
C04705=1034.687,-58.340,417.742,168.265,39.741,157.427
C04706=1034.693,-58.091,417.730,168.268,39.741,157.427
C04707=1034.700,-57.841,417.718,168.271,39.740,157.427
C04708=1034.707,-57.592,417.706,168.273,39.739,157.427
C04709=1034.713,-57.342,417.693,168.276,39.739,157.427
C04710=1034.719,-57.093,417.682,168.278,39.738,157.427
C04711=1034.725,-56.843,417.670,168.281,39.737,157.427
C04712=1034.731,-56.593,417.658,168.284,39.737,157.427
C04713=1034.738,-56.343,417.646,168.286,39.736,157.427
C04714=1034.744,-56.094,417.634,168.289,39.736,157.427
C04715=1034.750,-55.844,417.621,168.292,39.735,157.427
C04716=1034.757,-55.594,417.610,168.293,39.734,157.427
C04717=1034.763,-55.345,417.598,168.296,39.734,157.427
C04718=1034.769,-55.095,417.585,168.299,39.733,157.427
C04719=1034.775,-54.846,417.573,168.301,39.732,157.427
C04720=1034.782,-54.596,417.561,168.304,39.732,157.427
C04721=1034.789,-54.347,417.549,168.306,39.731,157.427
C04722=1034.795,-54.097,417.537,168.309,39.730,157.427
C04723=1034.801,-53.847,417.525,168.312,39.730,157.427
C04724=1034.808,-53.598,417.513,168.314,39.729,157.427
C04725=1034.814,-53.348,417.500,168.317,39.728,157.427
C04726=1034.820,-53.098,417.489,168.320,39.728,157.427
C04727=1034.827,-52.849,417.477,168.322,39.727,157.427
C04728=1034.832,-52.600,417.464,168.325,39.726,157.427
C04729=1034.839,-52.317,417.451,168.328,39.726,157.427
C04730=1034.847,-52.036,417.438,168.331,39.725,157.427
C04731=1034.854,-51.755,417.423,168.334,39.724,157.427
C04732=1034.861,-51.473,417.410,168.336,39.723,157.427
C04733=1034.868,-51.223,417.398,168.338,39.723,157.427
C04734=1034.874,-50.974,417.386,168.341,39.722,157.427
C04735=1034.880,-50.724,417.373,168.344,39.721,157.427
C04736=1034.887,-50.475,417.361,168.346,39.721,157.427
C04737=1034.893,-50.225,417.348,168.349,39.720,157.427
C04738=1034.899,-49.975,417.335,168.351,39.720,157.427
C04739=1034.906,-49.726,417.324,168.354,39.720,157.427
C04740=1034.912,-49.476,417.311,168.356,39.719,157.427
C04741=1034.918,-49.226,417.298,168.359,39.719,157.427
C04742=1034.924,-48.977,417.286,168.361,39.718,157.427
C04743=1034.930,-48.728,417.274,168.364,39.718,157.427
C04744=1034.936,-48.478,417.261,168.367,39.718,157.427
C04745=1034.942,-48.229,417.248,168.369,39.717,157.427
C04746=1034.949,-47.979,417.236,168.372,39.716,157.427
C04747=1034.954,-47.729,417.223,168.374,39.716,157.427
C04748=1034.960,-47.479,417.211,168.377,39.715,157.427
C04749=1034.967,-47.230,417.198,168.379,39.715,157.427
C04750=1034.973,-46.980,417.185,168.382,39.714,157.427
C04751=1034.979,-46.731,417.173,168.384,39.714,157.427
C04752=1034.986,-46.482,417.160,168.387,39.713,157.427
C04753=1034.992,-46.232,417.148,168.389,39.713,157.427
C04754=1034.998,-45.982,417.135,168.392,39.712,157.427
C04755=1035.004,-45.732,417.123,168.394,39.712,157.427
C04756=1035.011,-45.483,417.110,168.397,39.712,157.427
C04757=1035.017,-45.233,417.097,168.400,39.711,157.427
C04758=1035.023,-44.984,417.084,168.402,39.711,157.427
C04759=1035.029,-44.734,417.072,168.405,39.710,157.427
C04760=1035.035,-44.484,417.060,168.407,39.710,157.427
C04761=1035.042,-44.235,417.046,168.410,39.709,157.427
C04762=1035.048,-43.985,417.033,168.412,39.708,157.427
C04763=1035.055,-43.735,417.021,168.415,39.708,157.427
C04764=1035.061,-43.486,417.008,168.416,39.707,157.427
C04765=1035.067,-43.236,416.996,168.420,39.707,157.427
C04766=1035.073,-42.987,416.982,168.422,39.707,157.427
C04767=1035.080,-42.737,416.970,168.424,39.706,157.427
C04768=1035.086,-42.487,416.958,168.426,39.706,157.427
C04769=1035.092,-42.238,416.945,168.429,39.705,157.427
C04770=1035.098,-41.988,416.932,168.431,39.705,157.427
C04771=1035.105,-41.739,416.919,168.434,39.705,157.427
C04772=1035.111,-41.489,416.907,168.436,39.704,157.427
C04773=1035.117,-41.240,416.893,168.439,39.704,157.427
C04774=1035.123,-40.989,416.881,168.441,39.703,157.427
C04775=1035.130,-40.740,416.868,168.444,39.702,157.427
C04776=1035.136,-40.490,416.855,168.447,39.702,157.427
C04777=1035.142,-40.241,416.842,168.449,39.701,157.427
C04778=1035.148,-39.991,416.829,168.452,39.701,157.427
C04779=1035.155,-39.742,416.816,168.454,39.700,157.427
C04780=1035.161,-39.492,416.804,168.457,39.700,157.427
C04781=1035.168,-39.242,416.791,168.459,39.699,157.427
C04782=1035.174,-38.993,416.778,168.462,39.699,157.427
C04783=1035.180,-38.743,416.765,168.464,39.699,157.427
C04784=1035.186,-38.494,416.752,168.467,39.698,157.427
C04785=1035.192,-38.244,416.739,168.469,39.698,157.427
C04786=1035.199,-37.995,416.726,168.471,39.698,157.427
C04787=1035.205,-37.746,416.712,168.474,39.697,157.427
C04788=1035.211,-37.495,416.700,168.476,39.697,157.427
C04789=1035.217,-37.246,416.686,168.479,39.696,157.427
C04790=1035.224,-36.997,416.673,168.481,39.696,157.427
C04791=1035.230,-36.747,416.660,168.484,39.696,157.427
C04792=1035.236,-36.497,416.647,168.486,39.695,157.427
C04793=1035.243,-36.216,416.633,168.489,39.695,157.427
C04794=1035.251,-35.935,416.618,168.492,39.695,157.427
C04795=1035.257,-35.654,416.603,168.495,39.694,157.427
C04796=1035.264,-35.373,416.589,168.497,39.693,157.427
C04797=1035.270,-35.123,416.575,168.500,39.693,157.427
C04798=1035.277,-34.874,416.562,168.502,39.693,157.427
C04799=1035.283,-34.624,416.548,168.505,39.693,157.428
C04800=1035.289,-34.374,416.536,168.507,39.692,157.427
C04801=1035.296,-34.125,416.523,168.510,39.692,157.428
C04802=1035.302,-33.876,416.509,168.512,39.692,157.428
C04803=1035.308,-33.627,416.496,168.515,39.691,157.428
C04804=1035.315,-33.377,416.482,168.517,39.691,157.428
C04805=1035.321,-33.127,416.470,168.519,39.690,157.428
C04806=1035.327,-32.877,416.457,168.522,39.690,157.428
C04807=1035.333,-32.628,416.443,168.524,39.690,157.428
C04808=1035.339,-32.378,416.429,168.527,39.689,157.428
C04809=1035.345,-32.129,416.416,168.529,39.689,157.428
C04810=1035.351,-31.879,416.403,168.532,39.689,157.428
C04811=1035.358,-31.630,416.390,168.534,39.688,157.428
C04812=1035.364,-31.380,416.376,168.537,39.688,157.428
C04813=1035.371,-31.130,416.363,168.539,39.687,157.428
C04814=1035.377,-30.881,416.350,168.541,39.687,157.428
C04815=1035.384,-30.631,416.336,168.544,39.686,157.428
C04816=1035.390,-30.382,416.323,168.546,39.686,157.428
C04817=1035.396,-30.132,416.310,168.549,39.686,157.428
C04818=1035.403,-29.882,416.297,168.551,39.686,157.428
C04819=1035.409,-29.633,416.283,168.554,39.685,157.428
C04820=1035.415,-29.383,416.270,168.556,39.685,157.428
C04821=1035.422,-29.133,416.256,168.559,39.684,157.428
C04822=1035.428,-28.884,416.243,168.561,39.684,157.428
C04823=1035.434,-28.635,416.230,168.563,39.683,157.428
C04824=1035.441,-28.385,416.216,168.566,39.683,157.428
C04825=1035.447,-28.136,416.203,168.568,39.683,157.428
C04826=1035.453,-27.886,416.189,168.571,39.683,157.428
C04827=1035.460,-27.636,416.176,168.573,39.682,157.428
C04828=1035.466,-27.387,416.162,168.576,39.682,157.428
C04829=1035.472,-27.138,416.149,168.578,39.682,157.428
C04830=1035.479,-26.888,416.135,168.580,39.681,157.428
C04831=1035.485,-26.638,416.122,168.583,39.681,157.428
C04832=1035.490,-26.389,416.108,168.585,39.680,157.428
C04833=1035.497,-26.139,416.095,168.587,39.680,157.428
C04834=1035.504,-25.890,416.081,168.590,39.680,157.428
C04835=1035.509,-25.640,416.067,168.592,39.680,157.428
C04836=1035.516,-25.390,416.054,168.595,39.679,157.428
C04837=1035.522,-25.141,416.041,168.597,39.679,157.428
C04838=1035.528,-24.891,416.026,168.599,39.679,157.428
C04839=1035.535,-24.642,416.012,168.602,39.679,157.429
C04840=1035.541,-24.393,415.999,168.604,39.679,157.429
C04841=1035.547,-24.142,415.985,168.607,39.679,157.429
C04842=1035.553,-23.893,415.972,168.609,39.678,157.429
C04843=1035.559,-23.644,415.958,168.611,39.678,157.429
C04844=1035.565,-23.394,415.944,168.614,39.677,157.429
C04845=1035.572,-23.145,415.930,168.616,39.677,157.429
C04846=1035.579,-22.895,415.916,168.618,39.677,157.429
C04847=1035.584,-22.645,415.903,168.621,39.677,157.429
C04848=1035.591,-22.395,415.889,168.623,39.677,157.429
C04849=1035.597,-22.146,415.876,168.625,39.676,157.429
C04850=1035.603,-21.897,415.861,168.628,39.676,157.429
C04851=1035.610,-21.647,415.847,168.630,39.675,157.429
C04852=1035.616,-21.398,415.834,168.633,39.675,157.429
C04853=1035.622,-21.148,415.820,168.635,39.675,157.429
C04854=1035.628,-20.898,415.807,168.637,39.675,157.429
C04855=1035.635,-20.649,415.792,168.640,39.674,157.429
C04856=1035.641,-20.399,415.778,168.642,39.674,157.429
C04857=1035.648,-20.117,415.763,168.645,39.674,157.429
C04858=1035.655,-19.836,415.747,168.647,39.674,157.429
C04859=1035.663,-19.554,415.731,168.650,39.673,157.429
C04860=1035.669,-19.272,415.716,168.653,39.673,157.429
C04861=1035.676,-19.023,415.702,168.655,39.673,157.429
C04862=1035.683,-18.774,415.689,168.657,39.672,157.429
C04863=1035.689,-18.523,415.674,168.660,39.672,157.429
C04864=1035.695,-18.274,415.661,168.662,39.672,157.429
C04865=1035.701,-18.025,415.646,168.665,39.672,157.429
C04866=1035.708,-17.775,415.633,168.667,39.672,157.430
C04867=1035.714,-17.525,415.619,168.669,39.671,157.429
C04868=1035.721,-17.276,415.604,168.672,39.671,157.430
C04869=1035.727,-17.026,415.591,168.674,39.670,157.430
C04870=1035.734,-16.777,415.577,168.676,39.670,157.430
C04871=1035.739,-16.527,415.563,168.679,39.670,157.430
C04872=1035.746,-16.278,415.549,168.681,39.670,157.430
C04873=1035.752,-16.029,415.535,168.683,39.670,157.430
C04874=1035.759,-15.779,415.521,168.686,39.669,157.430
C04875=1035.765,-15.530,415.507,168.688,39.669,157.430
C04876=1035.771,-15.280,415.493,168.690,39.668,157.430
C04877=1035.778,-15.030,415.479,168.693,39.668,157.430
C04878=1035.784,-14.781,415.465,168.695,39.668,157.430
C04879=1035.790,-14.530,415.450,168.697,39.668,157.430
C04880=1035.797,-14.282,415.436,168.700,39.668,157.430
C04881=1035.803,-14.032,415.421,168.702,39.667,157.430
C04882=1035.809,-13.783,415.407,168.704,39.667,157.430
C04883=1035.816,-13.533,415.393,168.706,39.667,157.430
C04884=1035.821,-13.284,415.379,168.709,39.667,157.430
C04885=1035.828,-13.034,415.365,168.711,39.667,157.430
C04886=1035.834,-12.785,415.351,168.713,39.667,157.430
C04887=1035.840,-12.535,415.336,168.716,39.667,157.430
C04888=1035.847,-12.285,415.322,168.718,39.667,157.430
C04889=1035.853,-12.036,415.308,168.720,39.667,157.431
C04890=1035.859,-11.787,415.293,168.723,39.666,157.431
C04891=1035.865,-11.537,415.280,168.725,39.666,157.431
C04892=1035.872,-11.288,415.265,168.728,39.666,157.431
C04893=1035.878,-11.037,415.251,168.730,39.666,157.431
C04894=1035.884,-10.789,415.237,168.733,39.666,157.431
C04895=1035.891,-10.539,415.222,168.735,39.665,157.431
C04896=1035.897,-10.289,415.208,168.737,39.665,157.431
C04897=1035.903,-10.040,415.193,168.740,39.665,157.431
C04898=1035.909,-9.790,415.179,168.742,39.665,157.431
C04899=1035.916,-9.541,415.165,168.744,39.665,157.431
C04900=1035.922,-9.292,415.150,168.746,39.665,157.431
C04901=1035.928,-9.041,415.136,168.749,39.664,157.431
C04902=1035.935,-8.793,415.122,168.751,39.664,157.431
C04903=1035.941,-8.543,415.107,168.753,39.664,157.431
C04904=1035.948,-8.293,415.092,168.756,39.664,157.431
C04905=1035.954,-8.044,415.079,168.758,39.664,157.431
C04906=1035.960,-7.794,415.064,168.760,39.663,157.431
C04907=1035.967,-7.545,415.049,168.762,39.663,157.431
C04908=1035.973,-7.295,415.036,168.765,39.663,157.431
C04909=1035.979,-7.046,415.021,168.767,39.663,157.432
C04910=1035.986,-6.796,415.006,168.769,39.663,157.432
C04911=1035.993,-6.547,414.991,168.772,39.662,157.432
C04912=1035.998,-6.297,414.978,168.774,39.662,157.432
C04913=1036.005,-6.048,414.963,168.776,39.662,157.432
C04914=1036.012,-5.798,414.948,168.778,39.662,157.432
C04915=1036.017,-5.549,414.934,168.781,39.661,157.432
C04916=1036.024,-5.299,414.919,168.783,39.661,157.432
C04917=1036.031,-5.050,414.905,168.785,39.661,157.432
C04918=1036.037,-4.800,414.890,168.787,39.661,157.432
C04919=1036.043,-4.551,414.876,168.790,39.660,157.432
C04920=1036.050,-4.302,414.861,168.792,39.660,157.432
C04921=1036.057,-4.018,414.845,168.795,39.660,157.432
C04922=1036.064,-3.735,414.829,168.797,39.660,157.432
C04923=1036.071,-3.450,414.811,168.800,39.660,157.432
C04924=1036.078,-3.167,414.794,168.802,39.660,157.432
C04925=1036.084,-2.918,414.780,168.804,39.660,157.432
C04926=1036.091,-2.669,414.765,168.807,39.660,157.432
C04927=1036.097,-2.419,414.750,168.809,39.659,157.432
C04928=1036.103,-2.170,414.735,168.811,39.659,157.432
C04929=1036.109,-1.920,414.720,168.813,39.660,157.433
C04930=1036.115,-1.670,414.706,168.816,39.660,157.433
C04931=1036.122,-1.421,414.691,168.819,39.659,157.433
C04932=1036.127,-1.172,414.676,168.821,39.659,157.433
C04933=1036.134,-0.922,414.661,168.823,39.659,157.433
C04934=1036.140,-0.672,414.646,168.825,39.659,157.433
C04935=1036.147,-0.423,414.632,168.827,39.659,157.433
C04936=1036.153,-0.174,414.616,168.830,39.659,157.433
C04937=1036.159,0.075,414.601,168.832,39.659,157.433
C04938=1036.165,0.325,414.586,168.834,39.659,157.433
C04939=1036.172,0.575,414.571,168.836,39.659,157.433
C04940=1036.178,0.824,414.556,168.839,39.659,157.433
C04941=1036.184,1.073,414.542,168.841,39.659,157.433
C04942=1036.190,1.323,414.527,168.843,39.659,157.433
C04943=1036.197,1.573,414.512,168.845,39.658,157.434
C04944=1036.203,1.822,414.497,168.847,39.658,157.434
C04945=1036.209,2.072,414.482,168.850,39.658,157.434
C04946=1036.215,2.321,414.468,168.852,39.658,157.434
C04947=1036.222,2.571,414.453,168.854,39.658,157.434
C04948=1036.228,2.820,414.438,168.856,39.658,157.434
C04949=1036.234,3.070,414.423,168.858,39.658,157.434
C04950=1036.241,3.319,414.407,168.861,39.658,157.434
C04951=1036.247,3.568,414.392,168.863,39.658,157.434
C04952=1036.253,3.817,414.377,168.865,39.657,157.434
C04953=1036.260,4.067,414.363,168.868,39.658,157.434
C04954=1036.266,4.317,414.348,168.870,39.658,157.434
C04955=1036.272,4.566,414.333,168.872,39.658,157.434
C04956=1036.278,4.816,414.316,168.875,39.657,157.434
C04957=1036.285,5.065,414.301,168.877,39.657,157.434
C04958=1036.291,5.315,414.287,168.879,39.657,157.434
C04959=1036.297,5.564,414.272,168.881,39.657,157.434
C04960=1036.303,5.814,414.257,168.883,39.657,157.435
C04961=1036.310,6.063,414.241,168.886,39.657,157.435
C04962=1036.316,6.312,414.226,168.888,39.657,157.435
C04963=1036.323,6.562,414.211,168.890,39.657,157.435
C04964=1036.329,6.812,414.196,168.892,39.657,157.435
C04965=1036.336,7.061,414.182,168.894,39.656,157.435
C04966=1036.342,7.310,414.166,168.897,39.656,157.435
C04967=1036.349,7.560,414.151,168.899,39.656,157.435
C04968=1036.355,7.810,414.136,168.901,39.657,157.435
C04969=1036.361,8.059,414.121,168.903,39.656,157.435
C04970=1036.367,8.308,414.106,168.905,39.656,157.435
C04971=1036.374,8.557,414.091,168.908,39.656,157.435
C04972=1036.380,8.807,414.076,168.910,39.656,157.435
C04973=1036.386,9.056,414.060,168.912,39.656,157.435
C04974=1036.393,9.306,414.045,168.914,39.656,157.435
C04975=1036.399,9.556,414.030,168.916,39.655,157.435
C04976=1036.406,9.805,414.014,168.918,39.655,157.436
C04977=1036.412,10.054,413.999,168.921,39.656,157.436
C04978=1036.418,10.304,413.984,168.923,39.655,157.436
C04979=1036.425,10.553,413.968,168.926,39.655,157.436
C04980=1036.431,10.803,413.954,168.928,39.655,157.436
C04981=1036.438,11.052,413.939,168.930,39.655,157.436
C04982=1036.445,11.301,413.923,168.933,39.655,157.436
C04983=1036.451,11.551,413.908,168.935,39.655,157.436
C04984=1036.457,11.801,413.893,168.937,39.654,157.436
C04985=1036.464,12.067,413.876,168.939,39.654,157.436
C04986=1036.471,12.334,413.860,168.942,39.655,157.436
C04987=1036.478,12.601,413.843,168.944,39.654,157.436
C04988=1036.485,12.868,413.827,168.946,39.654,157.436
C04989=1036.493,13.192,413.807,168.949,39.654,157.436
C04990=1036.499,13.441,413.792,168.951,39.654,157.436
C04991=1036.506,13.690,413.776,168.953,39.654,157.436
C04992=1036.513,13.940,413.761,168.956,39.653,157.437
C04993=1036.519,14.189,413.746,168.958,39.653,157.437
C04994=1036.525,14.439,413.730,168.960,39.654,157.437
C04995=1036.532,14.688,413.714,168.962,39.654,157.437
C04996=1036.538,14.938,413.699,168.964,39.653,157.437
C04997=1036.544,15.187,413.683,168.966,39.653,157.437
C04998=1036.550,15.437,413.668,168.968,39.654,157.437
C04999=1036.557,15.686,413.653,168.970,39.654,157.437
C05000=1036.563,15.935,413.636,168.973,39.653,157.437
C05001=1036.569,16.185,413.621,168.975,39.653,157.437
C05002=1036.575,16.434,413.605,168.978,39.654,157.437
C05003=1036.582,16.684,413.590,168.980,39.654,157.437
C05004=1036.588,16.933,413.574,168.982,39.653,157.437
C05005=1036.594,17.183,413.559,168.984,39.653,157.437
C05006=1036.601,17.432,413.543,168.986,39.653,157.438
C05007=1036.607,17.681,413.528,168.989,39.653,157.438
C05008=1036.613,17.931,413.512,168.991,39.653,157.438
C05009=1036.620,18.180,413.496,168.993,39.653,157.438
C05010=1036.626,18.429,413.481,168.995,39.653,157.438
C05011=1036.633,18.680,413.465,168.997,39.653,157.438
C05012=1036.639,18.929,413.449,168.999,39.653,157.438
C05013=1036.645,19.178,413.433,169.001,39.653,157.438
C05014=1036.652,19.428,413.418,169.003,39.653,157.438
C05015=1036.658,19.677,413.402,169.006,39.653,157.438
C05016=1036.664,19.926,413.386,169.008,39.653,157.438
C05017=1036.671,20.176,413.371,169.010,39.653,157.438
C05018=1036.677,20.425,413.355,169.012,39.653,157.438
C05019=1036.683,20.674,413.339,169.014,39.653,157.438
C05020=1036.689,20.923,413.323,169.016,39.653,157.439
C05021=1036.696,21.174,413.308,169.018,39.653,157.439
C05022=1036.702,21.423,413.291,169.020,39.653,157.439
C05023=1036.709,21.672,413.276,169.023,39.653,157.439
C05024=1036.715,21.921,413.259,169.025,39.653,157.439
C05025=1036.721,22.171,413.245,169.028,39.653,157.439
C05026=1036.727,22.420,413.228,169.030,39.653,157.439
C05027=1036.734,22.669,413.213,169.032,39.653,157.439
C05028=1036.740,22.919,413.196,169.034,39.653,157.439
C05029=1036.747,23.169,413.180,169.036,39.653,157.439
C05030=1036.753,23.419,413.165,169.038,39.653,157.439
C05031=1036.759,23.668,413.149,169.040,39.653,157.439
C05032=1036.765,23.917,413.133,169.042,39.653,157.440
C05033=1036.772,24.166,413.117,169.044,39.653,157.440
C05034=1036.778,24.415,413.101,169.046,39.653,157.440
C05035=1036.785,24.664,413.085,169.048,39.653,157.440
C05036=1036.791,24.914,413.069,169.051,39.653,157.440
C05037=1036.797,25.164,413.053,169.053,39.653,157.440
C05038=1036.804,25.413,413.037,169.055,39.653,157.440
C05039=1036.810,25.663,413.021,169.057,39.653,157.440
C05040=1036.816,25.912,413.006,169.059,39.653,157.440
C05041=1036.823,26.162,412.989,169.062,39.653,157.440
C05042=1036.829,26.411,412.973,169.064,39.653,157.440
C05043=1036.835,26.660,412.957,169.066,39.653,157.440
C05044=1036.842,26.909,412.941,169.068,39.653,157.440
C05045=1036.848,27.159,412.925,169.070,39.653,157.440
C05046=1036.855,27.409,412.908,169.072,39.653,157.441
C05047=1036.861,27.658,412.893,169.075,39.653,157.441
C05048=1036.867,27.907,412.877,169.077,39.653,157.441
C05049=1036.874,28.194,412.859,169.079,39.653,157.441
C05050=1036.882,28.480,412.840,169.081,39.653,157.441
C05051=1036.890,28.767,412.821,169.084,39.653,157.441
C05052=1036.896,29.054,412.802,169.086,39.653,157.441
C05053=1036.903,29.303,412.787,169.088,39.653,157.441
C05054=1036.909,29.553,412.771,169.090,39.654,157.441
C05055=1036.915,29.802,412.754,169.092,39.654,157.441
C05056=1036.921,30.052,412.738,169.094,39.653,157.441
C05057=1036.928,30.300,412.721,169.097,39.654,157.442
C05058=1036.934,30.550,412.705,169.099,39.654,157.442
C05059=1036.940,30.799,412.689,169.102,39.653,157.442
C05060=1036.947,31.049,412.672,169.104,39.654,157.442
C05061=1036.953,31.299,412.656,169.106,39.654,157.442
C05062=1036.959,31.548,412.640,169.108,39.654,157.442
C05063=1036.965,31.797,412.624,169.110,39.654,157.442
C05064=1036.972,32.047,412.607,169.112,39.654,157.442
C05065=1036.978,32.296,412.591,169.114,39.654,157.442
C05066=1036.985,32.545,412.575,169.116,39.654,157.442
C05067=1036.991,32.794,412.558,169.118,39.654,157.442
C05068=1036.997,33.044,412.542,169.120,39.654,157.442
C05069=1037.003,33.294,412.526,169.122,39.654,157.443
C05070=1037.010,33.543,412.510,169.124,39.654,157.443
C05071=1037.016,33.793,412.493,169.126,39.654,157.443
C05072=1037.023,34.041,412.476,169.129,39.655,157.443
C05073=1037.029,34.291,412.460,169.131,39.654,157.443
C05074=1037.035,34.541,412.443,169.133,39.654,157.443
C05075=1037.042,34.790,412.428,169.135,39.655,157.443
C05076=1037.048,35.039,412.411,169.138,39.654,157.443
C05077=1037.055,35.289,412.394,169.140,39.654,157.443
C05078=1037.061,35.538,412.378,169.142,39.655,157.443
C05079=1037.067,35.787,412.362,169.144,39.655,157.443
C05080=1037.074,36.037,412.346,169.146,39.654,157.443
C05081=1037.080,36.286,412.329,169.148,39.655,157.444
C05082=1037.086,36.535,412.312,169.150,39.655,157.444
C05083=1037.093,36.785,412.296,169.152,39.655,157.444
C05084=1037.099,37.034,412.280,169.154,39.654,157.444
C05085=1037.106,37.283,412.263,169.156,39.655,157.444
C05086=1037.112,37.533,412.247,169.158,39.655,157.444
C05087=1037.118,37.782,412.230,169.161,39.655,157.444
C05088=1037.124,38.031,412.213,169.163,39.655,157.444
C05089=1037.131,38.281,412.197,169.165,39.655,157.444
C05090=1037.137,38.530,412.180,169.167,39.655,157.444
C05091=1037.143,38.779,412.163,169.169,39.655,157.444
C05092=1037.150,39.029,412.147,169.171,39.656,157.445
C05093=1037.156,39.279,412.131,169.173,39.656,157.445
C05094=1037.163,39.528,412.113,169.175,39.656,157.445
C05095=1037.168,39.777,412.097,169.177,39.656,157.445
C05096=1037.174,40.026,412.079,169.179,39.656,157.445
C05097=1037.181,40.276,412.063,169.181,39.656,157.445
C05098=1037.186,40.526,412.047,169.183,39.656,157.445
C05099=1037.193,40.774,412.030,169.185,39.657,157.445
C05100=1037.199,41.025,412.013,169.187,39.656,157.445
C05101=1037.206,41.273,411.996,169.189,39.656,157.445
C05102=1037.212,41.523,411.979,169.192,39.657,157.446
C05103=1037.218,41.772,411.962,169.194,39.656,157.446
C05104=1037.224,42.021,411.946,169.196,39.657,157.446
C05105=1037.231,42.271,411.929,169.198,39.657,157.446
C05106=1037.237,42.520,411.912,169.200,39.657,157.446
C05107=1037.244,42.770,411.895,169.202,39.657,157.446
C05108=1037.250,43.019,411.879,169.204,39.657,157.446
C05109=1037.256,43.268,411.862,169.206,39.657,157.446
C05110=1037.263,43.518,411.845,169.208,39.657,157.446
C05111=1037.268,43.767,411.828,169.210,39.658,157.446
C05112=1037.275,44.017,411.811,169.212,39.658,157.446
C05113=1037.282,44.303,411.791,169.216,39.658,157.447
C05114=1037.288,44.589,411.772,169.218,39.658,157.447
C05115=1037.296,44.876,411.753,169.220,39.658,157.447
C05116=1037.303,45.162,411.733,169.223,39.659,157.447
C05117=1037.309,45.413,411.716,169.225,39.659,157.447
C05118=1037.315,45.661,411.699,169.226,39.659,157.447
C05119=1037.322,45.910,411.682,169.228,39.659,157.447
C05120=1037.328,46.160,411.665,169.230,39.659,157.447
C05121=1037.334,46.409,411.648,169.232,39.659,157.447
C05122=1037.341,46.659,411.630,169.234,39.660,157.448
C05123=1037.347,46.908,411.614,169.236,39.660,157.448
C05124=1037.353,47.158,411.596,169.239,39.660,157.448
C05125=1037.359,47.406,411.579,169.241,39.660,157.448
C05126=1037.365,47.656,411.563,169.243,39.660,157.448
C05127=1037.371,47.905,411.545,169.245,39.660,157.448
C05128=1037.377,48.154,411.528,169.247,39.661,157.448
C05129=1037.384,48.404,411.511,169.249,39.661,157.448
C05130=1037.390,48.653,411.494,169.251,39.661,157.448
C05131=1037.396,48.903,411.476,169.253,39.661,157.449
C05132=1037.402,49.151,411.459,169.255,39.661,157.449
C05133=1037.409,49.401,411.443,169.257,39.661,157.449
C05134=1037.415,49.651,411.425,169.259,39.662,157.449
C05135=1037.421,49.900,411.408,169.261,39.661,157.449
C05136=1037.428,50.149,411.391,169.264,39.662,157.449
C05137=1037.434,50.398,411.373,169.266,39.662,157.449
C05138=1037.440,50.648,411.357,169.268,39.662,157.449
C05139=1037.447,50.897,411.339,169.270,39.662,157.449
C05140=1037.452,51.146,411.322,169.272,39.663,157.450
C05141=1037.459,51.396,411.305,169.274,39.662,157.450
C05142=1037.465,51.645,411.288,169.276,39.663,157.450
C05143=1037.471,51.895,411.270,169.278,39.663,157.450
C05144=1037.478,52.144,411.253,169.280,39.663,157.450
C05145=1037.484,52.393,411.236,169.282,39.663,157.450
C05146=1037.490,52.643,411.218,169.284,39.663,157.450
C05147=1037.497,52.891,411.201,169.286,39.663,157.450
C05148=1037.503,53.141,411.184,169.288,39.663,157.450
C05149=1037.509,53.390,411.167,169.291,39.664,157.450
C05150=1037.515,53.640,411.150,169.293,39.664,157.450
C05151=1037.522,53.889,411.133,169.295,39.664,157.451
C05152=1037.528,54.138,411.115,169.297,39.664,157.451
C05153=1037.535,54.388,411.097,169.299,39.664,157.451
C05154=1037.541,54.637,411.080,169.301,39.664,157.451
C05155=1037.547,54.886,411.062,169.303,39.665,157.451
C05156=1037.553,55.135,411.045,169.305,39.664,157.451
C05157=1037.560,55.385,411.029,169.307,39.664,157.451
C05158=1037.566,55.635,411.011,169.309,39.665,157.451
C05159=1037.572,55.884,410.994,169.311,39.665,157.451
C05160=1037.579,56.133,410.977,169.313,39.665,157.451
C05161=1037.585,56.382,410.959,169.315,39.665,157.451
C05162=1037.591,56.631,410.942,169.318,39.665,157.452
C05163=1037.598,56.881,410.924,169.320,39.665,157.452
C05164=1037.604,57.130,410.907,169.322,39.665,157.452
C05165=1037.611,57.379,410.889,169.324,39.666,157.452
C05166=1037.617,57.629,410.872,169.326,39.665,157.452
C05167=1037.623,57.878,410.855,169.328,39.666,157.452
C05168=1037.630,58.127,410.837,169.330,39.666,157.452
C05169=1037.636,58.377,410.819,169.332,39.666,157.452
C05170=1037.642,58.626,410.802,169.334,39.666,157.452
C05171=1037.649,58.875,410.785,169.336,39.666,157.452
C05172=1037.655,59.125,410.767,169.338,39.666,157.453
C05173=1037.662,59.374,410.750,169.340,39.666,157.453
C05174=1037.668,59.623,410.732,169.343,39.667,157.453
C05175=1037.675,59.873,410.715,169.345,39.666,157.453
C05176=1037.681,60.121,410.698,169.347,39.666,157.453
C05177=1037.688,60.408,410.677,169.349,39.667,157.453
C05178=1037.695,60.694,410.658,169.352,39.667,157.453
C05179=1037.703,60.981,410.637,169.354,39.667,157.453
C05180=1037.710,61.267,410.617,169.356,39.667,157.453
C05181=1037.717,61.516,410.600,169.358,39.667,157.453
C05182=1037.723,61.765,410.581,169.360,39.667,157.454
C05183=1037.730,62.015,410.564,169.362,39.667,157.454
C05184=1037.736,62.263,410.547,169.364,39.667,157.454
C05185=1037.742,62.513,410.529,169.366,39.667,157.454
C05186=1037.749,62.763,410.512,169.368,39.668,157.454
C05187=1037.755,63.012,410.494,169.370,39.668,157.454
C05188=1037.762,63.261,410.477,169.372,39.667,157.454
C05189=1037.768,63.510,410.459,169.375,39.668,157.454
C05190=1037.775,63.760,410.441,169.377,39.668,157.454
C05191=1037.782,64.009,410.423,169.379,39.668,157.454
C05192=1037.787,64.258,410.406,169.381,39.668,157.454
C05193=1037.793,64.508,410.388,169.383,39.669,157.455
C05194=1037.800,64.757,410.371,169.385,39.668,157.455
C05195=1037.807,65.006,410.352,169.387,39.669,157.455
C05196=1037.812,65.255,410.334,169.389,39.669,157.455
C05197=1037.819,65.505,410.317,169.391,39.669,157.455
C05198=1037.825,65.754,410.298,169.393,39.669,157.455
C05199=1037.831,66.003,410.281,169.395,39.669,157.455
C05200=1037.838,66.252,410.264,169.397,39.669,157.455
C05201=1037.844,66.502,410.246,169.400,39.670,157.455
C05202=1037.850,66.751,410.227,169.402,39.670,157.455
C05203=1037.857,67.001,410.210,169.404,39.670,157.456
C05204=1037.863,67.250,410.192,169.406,39.670,157.456
C05205=1037.869,67.499,410.173,169.408,39.670,157.456
C05206=1037.875,67.749,410.155,169.410,39.670,157.456
C05207=1037.882,67.998,410.138,169.412,39.671,157.456
C05208=1037.888,68.246,410.120,169.414,39.671,157.456
C05209=1037.894,68.496,410.102,169.416,39.671,157.456
C05210=1037.900,68.746,410.084,169.418,39.671,157.456
C05211=1037.907,68.995,410.066,169.419,39.671,157.456
C05212=1037.913,69.244,410.048,169.422,39.672,157.457
C05213=1037.919,69.493,410.030,169.424,39.672,157.457
C05214=1037.925,69.743,410.012,169.426,39.672,157.457
C05215=1037.932,69.992,409.993,169.428,39.672,157.457
C05216=1037.939,70.241,409.976,169.430,39.672,157.457
C05217=1037.944,70.490,409.958,169.432,39.672,157.457
C05218=1037.951,70.739,409.940,169.434,39.673,157.457
C05219=1037.957,70.989,409.922,169.436,39.673,157.457
C05220=1037.963,71.238,409.903,169.438,39.673,157.457
C05221=1037.969,71.488,409.885,169.440,39.674,157.458
C05222=1037.975,71.736,409.867,169.443,39.673,157.458
C05223=1037.982,71.986,409.849,169.445,39.674,157.458
C05224=1037.988,72.235,409.831,169.447,39.674,157.458
C05225=1037.995,72.485,409.813,169.449,39.674,157.458
C05226=1038.001,72.734,409.794,169.451,39.675,157.458
C05227=1038.007,72.984,409.776,169.453,39.675,157.458
C05228=1038.013,73.232,409.758,169.455,39.675,157.458
C05229=1038.019,73.482,409.740,169.457,39.675,157.458
C05230=1038.026,73.731,409.721,169.459,39.675,157.459
C05231=1038.032,73.980,409.703,169.461,39.675,157.459
C05232=1038.039,74.229,409.685,169.463,39.676,157.459
C05233=1038.045,74.478,409.667,169.466,39.676,157.459
C05234=1038.051,74.727,409.649,169.467,39.676,157.459
C05235=1038.057,74.977,409.631,169.469,39.676,157.459
C05236=1038.064,75.226,409.612,169.471,39.676,157.459
C05237=1038.070,75.475,409.594,169.473,39.677,157.459
C05238=1038.076,75.725,409.575,169.475,39.677,157.459
C05239=1038.082,75.974,409.557,169.477,39.677,157.460
C05240=1038.089,76.223,409.539,169.479,39.678,157.460
C05241=1038.096,76.509,409.518,169.482,39.677,157.460
C05242=1038.103,76.795,409.496,169.484,39.678,157.460
C05243=1038.111,77.082,409.476,169.486,39.678,157.460
C05244=1038.117,77.367,409.455,169.489,39.678,157.460
C05245=1038.124,77.616,409.436,169.491,39.679,157.460
C05246=1038.130,77.866,409.418,169.493,39.678,157.460
C05247=1038.136,78.115,409.400,169.495,39.679,157.461
C05248=1038.143,78.364,409.381,169.497,39.679,157.461
C05249=1038.149,78.614,409.362,169.499,39.679,157.461
C05250=1038.155,78.863,409.344,169.501,39.680,157.461
C05251=1038.161,79.112,409.326,169.503,39.680,157.461
C05252=1038.167,79.361,409.307,169.505,39.680,157.461
C05253=1038.173,79.610,409.288,169.508,39.680,157.461
C05254=1038.180,79.859,409.270,169.510,39.681,157.461
C05255=1038.186,80.109,409.252,169.512,39.681,157.462
C05256=1038.192,80.358,409.233,169.514,39.681,157.462
C05257=1038.198,80.607,409.214,169.515,39.682,157.462
C05258=1038.204,80.857,409.195,169.517,39.682,157.462
C05259=1038.211,81.106,409.176,169.519,39.682,157.462
C05260=1038.217,81.355,409.158,169.521,39.683,157.462
C05261=1038.223,81.605,409.140,169.523,39.682,157.462
C05262=1038.230,81.854,409.121,169.526,39.683,157.462
C05263=1038.235,82.102,409.103,169.528,39.683,157.462
C05264=1038.241,82.352,409.084,169.530,39.683,157.463
C05265=1038.248,82.601,409.065,169.532,39.684,157.463
C05266=1038.254,82.850,409.046,169.534,39.683,157.463
C05267=1038.260,83.099,409.028,169.536,39.684,157.463
C05268=1038.266,83.349,409.010,169.538,39.684,157.463
C05269=1038.272,83.598,408.991,169.540,39.684,157.463
C05270=1038.279,83.847,408.972,169.542,39.685,157.463
C05271=1038.285,84.097,408.953,169.545,39.685,157.464
C05272=1038.291,84.346,408.935,169.547,39.685,157.464
C05273=1038.298,84.595,408.916,169.549,39.686,157.464
C05274=1038.304,84.844,408.897,169.551,39.685,157.464
C05275=1038.310,85.093,408.878,169.553,39.686,157.464
C05276=1038.316,85.343,408.859,169.555,39.686,157.464
C05277=1038.323,85.592,408.841,169.557,39.686,157.464
C05278=1038.329,85.841,408.822,169.558,39.687,157.464
C05279=1038.335,86.090,408.803,169.560,39.687,157.464
C05280=1038.341,86.339,408.784,169.562,39.687,157.465
C05281=1038.348,86.588,408.766,169.565,39.687,157.465
C05282=1038.354,86.838,408.747,169.567,39.687,157.465
C05283=1038.361,87.087,408.728,169.569,39.688,157.465
C05284=1038.366,87.336,408.709,169.571,39.688,157.465
C05285=1038.373,87.585,408.690,169.573,39.688,157.465
C05286=1038.379,87.834,408.672,169.575,39.689,157.465
C05287=1038.386,88.083,408.653,169.577,39.688,157.465
C05288=1038.393,88.333,408.634,169.579,39.689,157.465
C05289=1038.398,88.583,408.615,169.581,39.689,157.466
C05290=1038.405,88.832,408.596,169.583,39.689,157.466
C05291=1038.411,89.081,408.578,169.586,39.690,157.466
C05292=1038.418,89.330,408.559,169.588,39.689,157.466
C05293=1038.423,89.580,408.540,169.590,39.690,157.466
C05294=1038.430,89.829,408.521,169.592,39.690,157.466
C05295=1038.436,90.078,408.502,169.594,39.690,157.466
C05296=1038.442,90.327,408.483,169.596,39.691,157.466
C05297=1038.449,90.576,408.464,169.598,39.691,157.467
C05298=1038.455,90.825,408.445,169.600,39.691,157.467
C05299=1038.461,91.074,408.426,169.602,39.691,157.467
C05300=1038.467,91.323,408.407,169.605,39.692,157.467
C05301=1038.473,91.573,408.388,169.607,39.692,157.467
C05302=1038.480,91.821,408.369,169.609,39.692,157.467
C05303=1038.486,92.071,408.349,169.611,39.693,157.467
C05304=1038.492,92.321,408.330,169.612,39.693,157.468
C05305=1038.498,92.607,408.309,169.615,39.694,157.468
C05306=1038.505,92.892,408.286,169.617,39.694,157.468
C05307=1038.513,93.179,408.265,169.619,39.694,157.468
C05308=1038.520,93.464,408.242,169.621,39.694,157.468
C05309=1038.526,93.713,408.224,169.624,39.695,157.468
C05310=1038.532,93.963,408.204,169.626,39.695,157.468
C05311=1038.539,94.211,408.185,169.628,39.695,157.468
C05312=1038.545,94.461,408.166,169.630,39.696,157.469
C05313=1038.552,94.711,408.147,169.632,39.696,157.469
C05314=1038.557,94.960,408.127,169.634,39.696,157.469
C05315=1038.564,95.208,408.108,169.636,39.696,157.469
C05316=1038.570,95.458,408.089,169.638,39.697,157.469
C05317=1038.575,95.707,408.070,169.640,39.697,157.469
C05318=1038.582,95.956,408.050,169.643,39.697,157.469
C05319=1038.588,96.205,408.031,169.645,39.698,157.470
C05320=1038.595,96.455,408.012,169.647,39.698,157.470
C05321=1038.601,96.704,407.992,169.649,39.698,157.470
C05322=1038.607,96.953,407.973,169.651,39.698,157.470
C05323=1038.613,97.202,407.954,169.653,39.699,157.470
C05324=1038.620,97.451,407.935,169.655,39.699,157.470
C05325=1038.625,97.700,407.916,169.657,39.699,157.470
C05326=1038.633,97.950,407.896,169.660,39.700,157.470
C05327=1038.638,98.199,407.877,169.662,39.700,157.471
C05328=1038.645,98.448,407.858,169.664,39.700,157.471
C05329=1038.651,98.697,407.838,169.666,39.701,157.471
C05330=1038.657,98.946,407.819,169.668,39.700,157.471
C05331=1038.664,99.196,407.799,169.670,39.701,157.471
C05332=1038.670,99.445,407.780,169.672,39.701,157.471
C05333=1038.676,99.694,407.761,169.674,39.701,157.471
C05334=1038.683,99.943,407.742,169.676,39.702,157.471
C05335=1038.688,100.192,407.722,169.679,39.702,157.472
C05336=1038.695,100.442,407.702,169.681,39.702,157.472
C05337=1038.701,100.691,407.683,169.683,39.702,157.472
C05338=1038.707,100.940,407.664,169.684,39.703,157.472
C05339=1038.713,101.189,407.644,169.686,39.703,157.472
C05340=1038.719,101.438,407.624,169.688,39.704,157.472
C05341=1038.725,101.687,407.604,169.690,39.704,157.472
C05342=1038.732,101.936,407.585,169.692,39.704,157.473
C05343=1038.738,102.185,407.565,169.694,39.705,157.473
C05344=1038.744,102.435,407.546,169.697,39.705,157.473
C05345=1038.750,102.684,407.526,169.699,39.706,157.473
C05346=1038.756,102.934,407.507,169.701,39.705,157.473
C05347=1038.763,103.182,407.487,169.703,39.706,157.473
C05348=1038.769,103.431,407.467,169.705,39.706,157.473
C05349=1038.774,103.680,407.448,169.707,39.707,157.474
C05350=1038.780,103.929,407.428,169.709,39.707,157.474
C05351=1038.787,104.179,407.408,169.711,39.707,157.474
C05352=1038.793,104.428,407.389,169.714,39.708,157.474
C05353=1038.799,104.677,407.369,169.716,39.708,157.474
C05354=1038.805,104.925,407.349,169.718,39.708,157.474
C05355=1038.812,105.176,407.330,169.720,39.709,157.474
C05356=1038.818,105.424,407.310,169.722,39.709,157.474
C05357=1038.825,105.673,407.290,169.724,39.709,157.475
C05358=1038.830,105.922,407.271,169.726,39.710,157.475
C05359=1038.837,106.172,407.251,169.729,39.710,157.475
C05360=1038.843,106.421,407.231,169.731,39.710,157.475
C05361=1038.848,106.670,407.211,169.733,39.710,157.475
C05362=1038.855,106.920,407.191,169.735,39.711,157.475
C05363=1038.862,107.168,407.172,169.737,39.711,157.476
C05364=1038.867,107.418,407.153,169.739,39.711,157.476
C05365=1038.874,107.667,407.132,169.741,39.712,157.476
C05366=1038.880,107.916,407.112,169.743,39.712,157.476
C05367=1038.886,108.165,407.092,169.745,39.713,157.476
C05368=1038.892,108.414,407.073,169.747,39.712,157.476
C05369=1038.900,108.701,407.050,169.750,39.713,157.476
C05370=1038.907,108.986,407.027,169.752,39.713,157.476
C05371=1038.914,109.272,407.004,169.755,39.714,157.477
C05372=1038.921,109.558,406.981,169.757,39.714,157.477
C05373=1038.927,109.807,406.963,169.759,39.715,157.477
C05374=1038.934,110.056,406.942,169.761,39.715,157.477
C05375=1038.940,110.305,406.922,169.763,39.715,157.477
C05376=1038.947,110.555,406.902,169.766,39.716,157.477
C05377=1038.953,110.803,406.882,169.768,39.716,157.478
C05378=1038.959,111.052,406.862,169.770,39.716,157.478
C05379=1038.965,111.302,406.842,169.772,39.716,157.478
C05380=1038.971,111.551,406.823,169.774,39.717,157.478
C05381=1038.977,111.800,406.803,169.776,39.717,157.478
C05382=1038.983,112.050,406.782,169.778,39.718,157.478
C05383=1038.989,112.298,406.762,169.781,39.718,157.478
C05384=1038.995,112.547,406.742,169.783,39.719,157.479
C05385=1039.002,112.797,406.722,169.785,39.718,157.479
C05386=1039.008,113.045,406.702,169.787,39.719,157.479
C05387=1039.014,113.294,406.682,169.789,39.719,157.479
C05388=1039.021,113.544,406.662,169.791,39.720,157.479
C05389=1039.027,113.793,406.642,169.793,39.720,157.479
C05390=1039.032,114.042,406.621,169.795,39.721,157.479
C05391=1039.038,114.291,406.601,169.798,39.721,157.480
C05392=1039.044,114.540,406.581,169.800,39.722,157.480
C05393=1039.051,114.790,406.561,169.802,39.722,157.480
C05394=1039.056,115.039,406.540,169.804,39.723,157.480
C05395=1039.062,115.288,406.520,169.806,39.723,157.480
C05396=1039.069,115.537,406.500,169.808,39.723,157.480
C05397=1039.075,115.786,406.480,169.810,39.723,157.481
C05398=1039.080,116.035,406.459,169.813,39.724,157.481
C05399=1039.087,116.284,406.438,169.815,39.724,157.481
C05400=1039.093,116.533,406.418,169.817,39.725,157.481
C05401=1039.099,116.781,406.398,169.818,39.725,157.481
C05402=1039.105,117.031,406.378,169.820,39.726,157.481
C05403=1039.111,117.280,406.358,169.822,39.726,157.482
C05404=1039.117,117.530,406.337,169.824,39.727,157.482
C05405=1039.123,117.779,406.317,169.827,39.727,157.482
C05406=1039.129,118.028,406.297,169.829,39.728,157.482
C05407=1039.136,118.276,406.276,169.831,39.728,157.482
C05408=1039.142,118.525,406.256,169.833,39.729,157.482
C05409=1039.147,118.775,406.235,169.835,39.729,157.483
C05410=1039.153,119.024,406.215,169.837,39.730,157.483
C05411=1039.160,119.273,406.195,169.840,39.730,157.483
C05412=1039.166,119.522,406.173,169.842,39.730,157.483
C05413=1039.172,119.771,406.153,169.844,39.730,157.483
C05414=1039.178,120.020,406.133,169.846,39.731,157.483
C05415=1039.184,120.269,406.113,169.848,39.731,157.483
C05416=1039.190,120.519,406.092,169.851,39.732,157.484
C05417=1039.196,120.767,406.071,169.853,39.732,157.484
C05418=1039.203,121.017,406.051,169.856,39.733,157.484
C05419=1039.208,121.266,406.031,169.858,39.733,157.484
C05420=1039.215,121.515,406.010,169.860,39.733,157.484
C05421=1039.221,121.763,405.990,169.862,39.734,157.484
C05422=1039.228,122.013,405.969,169.864,39.734,157.485
C05423=1039.233,122.262,405.949,169.866,39.735,157.485
C05424=1039.240,122.512,405.928,169.868,39.735,157.485
C05425=1039.246,122.760,405.908,169.870,39.735,157.485
C05426=1039.252,123.010,405.887,169.873,39.736,157.485
C05427=1039.258,123.258,405.867,169.875,39.736,157.485
C05428=1039.265,123.507,405.846,169.877,39.737,157.486
C05429=1039.270,123.756,405.825,169.879,39.737,157.486
C05430=1039.276,124.006,405.805,169.881,39.737,157.486
C05431=1039.283,124.254,405.784,169.883,39.738,157.486
C05432=1039.289,124.504,405.763,169.886,39.738,157.486
C05433=1039.296,124.789,405.740,169.888,39.739,157.486
C05434=1039.303,125.075,405.716,169.891,39.739,157.487
C05435=1039.310,125.362,405.693,169.893,39.740,157.487
C05436=1039.317,125.647,405.669,169.895,39.740,157.487
C05437=1039.324,125.896,405.648,169.897,39.741,157.487
C05438=1039.330,126.145,405.628,169.899,39.741,157.487
C05439=1039.336,126.394,405.607,169.902,39.741,157.487
C05440=1039.343,126.643,405.586,169.905,39.741,157.487
C05441=1039.349,126.892,405.566,169.907,39.742,157.488
C05442=1039.355,127.141,405.544,169.909,39.742,157.488
C05443=1039.361,127.390,405.524,169.911,39.743,157.488
C05444=1039.368,127.639,405.503,169.913,39.743,157.488
C05445=1039.373,127.889,405.483,169.915,39.744,157.488
C05446=1039.379,128.138,405.463,169.918,39.744,157.488
C05447=1039.386,128.387,405.442,169.920,39.745,157.489
C05448=1039.392,128.636,405.421,169.922,39.744,157.489
C05449=1039.399,128.885,405.400,169.924,39.745,157.489
C05450=1039.405,129.134,405.380,169.926,39.745,157.489
C05451=1039.411,129.383,405.358,169.928,39.746,157.489
C05452=1039.417,129.632,405.338,169.930,39.746,157.489
C05453=1039.424,129.881,405.317,169.934,39.747,157.490
C05454=1039.429,130.130,405.296,169.936,39.747,157.490
C05455=1039.436,130.379,405.275,169.938,39.748,157.490
C05456=1039.442,130.628,405.254,169.940,39.747,157.490
C05457=1039.448,130.877,405.234,169.942,39.748,157.490
C05458=1039.455,131.126,405.213,169.944,39.748,157.490
C05459=1039.461,131.376,405.192,169.946,39.749,157.490
C05460=1039.467,131.624,405.171,169.948,39.749,157.491
C05461=1039.474,131.873,405.150,169.951,39.750,157.491
C05462=1039.480,132.123,405.129,169.953,39.750,157.491
C05463=1039.485,132.372,405.107,169.955,39.751,157.491
C05464=1039.492,132.620,405.086,169.957,39.752,157.491
C05465=1039.497,132.870,405.066,169.959,39.752,157.492
C05466=1039.503,133.119,405.044,169.963,39.753,157.492
